(* PLC project TemplatePLC210_01, CODESYS CODESYS V3.5 SP17 Patch 3 *)
(* stored: creationDateTime 2025-07-22T12:00:36.9424136, version 3.5.14.30, modificationDateTime 2025-07-22T12:00:25.3757324, organization Production association OWEN *)

TYPE TRG_LeftSide :
STRUCT
	xFastDi01:				BOOL;
	xFastDi02:				BOOL;
	xFastDi03:				BOOL;
	xFastDi04:				BOOL;
	xFastDi05:				BOOL;
	xFastDi06:				BOOL;
	xFastDi07:				BOOL;
	xFastDi08:				BOOL;
	xFastDi09: 				BOOL;
	xFastDi10:				BOOL;
	xFastDi11:				BOOL;
	xFastDi12:				BOOL;
	
	xDo01:					BOOL;
	xDo02:					BOOL;
	xDo03:					BOOL;
	xDo04:					BOOL;
	
	udiCounterFastDi01:		UDINT;
	udiCounterFastDi02:		UDINT;
	udiCounterFastDi03:		UDINT;
	udiCounterFastDi04:		UDINT;
	udiCounterFastDi05:		UDINT;
	udiCounterFastDi06:		UDINT;
	udiCounterFastDi07:		UDINT;
	udiCounterFastDi08:		UDINT;
	udiCounterFastDi09:		UDINT;
	udiCounterFastDi10:		UDINT;
	udiCounterFastDi11:		UDINT;
	udiCounterFastDi12:		UDINT;
	
	udiPulseDurationFastDi01:	UDINT;
	udiPulseDurationFastDi02:	UDINT;
	udiPulseDurationFastDi03:	UDINT;
	udiPulseDurationFastDi04:	UDINT;
	udiPulseDurationFastDi05:	UDINT;
	udiPulseDurationFastDi06:	UDINT;
	udiPulseDurationFastDi07:	UDINT;
	udiPulseDurationFastDi08:	UDINT;
	udiPulseDurationFastDi09:	UDINT;
	udiPulseDurationFastDi10:	UDINT;
	udiPulseDurationFastDi11:	UDINT;
	udiPulseDurationFastDi12:	UDINT;

	udiPulsePeriodFastDi01:		UDINT;
	udiPulsePeriodFastDi02:		UDINT;
	udiPulsePeriodFastDi03:		UDINT;
	udiPulsePeriodFastDi04:		UDINT;
	udiPulsePeriodFastDi05:		UDINT;
	udiPulsePeriodFastDi06:		UDINT;
	udiPulsePeriodFastDi07:		UDINT;
	udiPulsePeriodFastDi08:		UDINT;
	udiPulsePeriodFastDi09:		UDINT;
	udiPulsePeriodFastDi10:		UDINT;
	udiPulsePeriodFastDi11:		UDINT;
	udiPulsePeriodFastDi12:		UDINT;
	
	udiGenPulseCountDo01:	    UDINT;
	udiGenPulseCountDo02:	    UDINT;
	udiGenPulseCountDo03:	    UDINT;
	udiGenPulseCountDo04:	    UDINT;
	
	udiGenPulseCountLeftDo01:	UDINT;
	udiGenPulseCountLeftDo02:	UDINT;
	udiGenPulseCountLeftDo03:	UDINT;
	udiGenPulseCountLeftDo04:	UDINT;
	
	udiPwmDutyCycleDo01:		UDINT;
	udiPwmDutyCycleDo02:		UDINT;
	udiPwmDutyCycleDo03:		UDINT;
	udiPwmDutyCycleDo04:		UDINT;
	
	diPulseCounterAbEncoder01: DINT;
	diPulseCounterAbEncoder02: DINT;
	diPulseCounterAbEncoder03: DINT;
	diPulseCounterAbEncoder04: DINT;
	diPulseCounterAbEncoder05: DINT;
	diPulseCounterAbEncoder06: DINT;
	
	diPulseCounterAbzEncoder01: DINT;
	diPulseCounterAbzEncoder02: DINT;
	diPulseCounterAbzEncoder03: DINT;
	
	diTurnCounterAbzEncoder01: DINT;
	diTurnCounterAbzEncoder02: DINT;
	diTurnCounterAbzEncoder03: DINT;
END_STRUCT
END_TYPE

TYPE TRG_Debug :
STRUCT
	xEnable: 			BOOL;
	udiPollingTime:		UDINT;
	udiRamUsedSize:		UDINT;
	udiRamFreeSize:		UDINT;
	udiCountHandles:	UDINT;
	udiProcUsage:		UDINT;
END_STRUCT
END_TYPE

TYPE TRG_Drives :
STRUCT
	xEnable:			BOOL;
	
	uliFsFullSize: 		ULINT;
	uliFsUsedSize: 		ULINT;
	uliFsFreeSize: 		ULINT;
	
	xUsbMounted:		BOOL;
	xUsbUnmount:		BOOL;
	xUsbUnmountDone:	BOOL;
	
	uliUsbFullSize: 	ULINT;
	uliUsbUsedSize: 	ULINT;
	uliUsbFreeSize: 	ULINT;
	
	xSdMounted:			BOOL;
	xSdUnmount:			BOOL;
	xSdUnmountDone:		BOOL;
	
	uliSdFullSize: 		ULINT;
	uliSdUsedSize: 		ULINT;
	uliSdFreeSize: 		ULINT;
END_STRUCT
END_TYPE

TYPE TRG_Info :
STRUCT
	sVendorName: 			STRING;
	sDeviceName: 			STRING;
	sSerialId: 				STRING;
	sRuntimeVersion:		STRING;
	sFirmwareVersion: 		STRING;
	sLinuxVersion: 			STRING;
	sNeedTargetVersion:		STRING;
	
	sProjectName:			STRING;
	sAuthorName:			STRING;
	sProjectVersion:		STRING;
	sProjectProfile:		STRING;
	dtProjectLastChanges:	DT;
END_STRUCT
END_TYPE

TYPE TRG_PLC210 :
STRUCT
	xPowerInput1:	  BOOL;
	xPowerInput2: 	  BOOL;
	xServiceButton:   BOOL;
	rCpuTemp:		  REAL;
	xStartStopSwitch: BOOL;
END_STRUCT
END_TYPE

TYPE TRG_RTC :
STRUCT
	uiGetYear:			UINT;
	usiGetMonth:		USINT;
	usiGetDay:			USINT;
	usiGetHour:			USINT;
	usiGetMinute:		USINT;
	usiGetSecond:		USINT;
	usiGetDayOfWeek:	USINT;
	usiGetWeekOfYear:	USINT;
	sGetFormatDate:		STRING;
	sGetFormatTime:		STRING;
	siGetUtcOffset:		SINT;
	dtDateAndTime:		DT;
	
	
	uiSetYear:			UINT;
	usiSetMonth:		USINT;
	usiSetDay:			USINT;
	usiSetHour:			USINT;
	usiSetMinute:		USINT;
	usiSetSecond:		USINT;
	siSetUtcOffset:		SINT;
	xUpdateSettings:	BOOL;
	
	xEnableNtp:			BOOL;
	xIsNtpEnabled:		BOOL;
	sPreferNtpServer:	STRING;
	usiNtpErrorCode:	USINT;
	
	ltSystemTick:		LTIME;
END_STRUCT
END_TYPE

TYPE TRG_Watchdog :
STRUCT
	eHandlingType:						Watchdog.ExceptionHandling;
	udiLastExceptionCode:				UDINT;
	sLastExceptionText:					STRING;
	dtLastExceptionTime:				DT;
	xIsHardwareWatchdogReboot:			BOOL;
	xDoReboot:							BOOL;
	usiPowerRebootCount:				USINT;
	usiExceptionRebootCount:			USINT;
	usiCommandRebootCount:				USINT;
	usiHardwareWatchdogRebootCount:		USINT;
	xResetCounters:						BOOL;
END_STRUCT
END_TYPE

TYPE TRG_RightSide :
STRUCT
	xSystemBusLink:				  BOOL;
	udiSystemBusError:  		  UDINT;
	
	xDo05:						  BOOL;
	xDo06:						  BOOL;
	xDo07:						  BOOL;
	xDo08:						  BOOL;
	xDo09:						  BOOL;
	xDo10:						  BOOL;
	xDo11:						  BOOL;
	xDo12:						  BOOL;

	xWriteAllAiSettings:  		  BOOL;
	
	xWriteSettingsAi1:	  		  BOOL;
	eWriteSensorTypeAi1:		  Mx210Assistant.ANALOG_SENSORS;
	rWriteOffsetAi1:			  REAL;
	rWriteMulAi1:			 	  REAL;
	rWriteHighLimitAi1:		 	  REAL;
	rWriteLowLimitAi1:		 	  REAL;
	uiWriteFilterBandAi1:	  	  UINT;
	uiWriteFilterTimeAi1:	  	  UINT;
	
	xWriteSettingsAi2:	  		  BOOL;
	eWriteSensorTypeAi2:		  Mx210Assistant.ANALOG_SENSORS;
	rWriteOffsetAi2:			  REAL;
	rWriteMulAi2:			 	  REAL;
	rWriteHighLimitAi2:		  	  REAL;
	rWriteLowLimitAi2:		  	  REAL;
	uiWriteFilterBandAi2:	  	  UINT;
	uiWriteFilterTimeAi2:	  	  UINT;
	
	xWriteSettingsAi3:	  		  BOOL;
	eWriteSensorTypeAi3:		  Mx210Assistant.ANALOG_SENSORS;
	rWriteOffsetAi3:			  REAL;
	rWriteMulAi3:			 	  REAL;
	rWriteHighLimitAi3:		  	  REAL;
	rWriteLowLimitAi3:		  	  REAL;
	uiWriteFilterBandAi3:	  	  UINT;
	uiWriteFilterTimeAi3:	  	  UINT;
	
	xWriteSettingsAi4:	  		  BOOL;
	eWriteSensorTypeAi4:		  Mx210Assistant.ANALOG_SENSORS;
	rWriteOffsetAi4:			  REAL;
	rWriteMulAi4:			 	  REAL;
	rWriteHighLimitAi4:		  	  REAL;
	rWriteLowLimitAi4:		  	  REAL;
	uiWriteFilterBandAi4:	  	  UINT;
	uiWriteFilterTimeAi4:	  	  UINT;
	
	xReadAllAiSettings:  		  BOOL;
	
	xReadSettingsAi1:	  		  BOOL;
	eReadSensorTypeAi1:		  	  Mx210Assistant.ANALOG_SENSORS;
	rReadOffsetAi1:			  	  REAL;
	rReadMulAi1:			 	  REAL;
	rReadHighLimitAi1:		 	  REAL;
	rReadLowLimitAi1:		 	  REAL;
	uiReadFilterBandAi1:	  	  UINT;
	uiReadFilterTimeAi1:	  	  UINT;
	
	xReadSettingsAi2:	  		  BOOL;
	eReadSensorTypeAi2:		  	  Mx210Assistant.ANALOG_SENSORS;
	rReadOffsetAi2:			  	  REAL;
	rReadMulAi2:			 	  REAL;
	rReadHighLimitAi2:		  	  REAL;
	rReadLowLimitAi2:		  	  REAL;
	uiReadFilterBandAi2:	  	  UINT;
	uiReadFilterTimeAi2:	  	  UINT;
	
	xReadSettingsAi3:	  		  BOOL;
	eReadSensorTypeAi3:		  	  Mx210Assistant.ANALOG_SENSORS;
	rReadOffsetAi3:			  	  REAL;
	rReadMulAi3:			 	  REAL;
	rReadHighLimitAi3:		  	  REAL;
	rReadLowLimitAi3:		  	  REAL;
	uiReadFilterBandAi3:	  	  UINT;
	uiReadFilterTimeAi3:	  	  UINT;
	
	xReadSettingsAi4:	  		  BOOL;
	eReadSensorTypeAi4:		  	  Mx210Assistant.ANALOG_SENSORS;
	rReadOffsetAi4:			  	  REAL;
	rReadMulAi4:			 	  REAL;
	rReadHighLimitAi4:		  	  REAL;
	rReadLowLimitAi4:		  	  REAL;
	uiReadFilterBandAi4:	  	  UINT;
	uiReadFilterTimeAi4:	  	  UINT;
	
	rValueAi1:					  REAL;
	uiTimeAi1:					  UINT;
	eStatusAi1:					  Mx210Assistant.ANALOG_SENSOR_ERRORS;
	
	rValueAi2:					  REAL;
	uiTimeAi2:					  UINT;
	eStatusAi2:					  Mx210Assistant.ANALOG_SENSOR_ERRORS;

	rValueAi3:					  REAL;
	uiTimeAi3:					  UINT;
	eStatusAi3:					  Mx210Assistant.ANALOG_SENSOR_ERRORS;

	rValueAi4:					  REAL;
	uiTimeAi4:					  UINT;
	eStatusAi4:					  Mx210Assistant.ANALOG_SENSOR_ERRORS;	
END_STRUCT
END_TYPE

TYPE TRG_Buzzer :
STRUCT
	xGet:	BOOL;
	xSet:	BOOL;
END_STRUCT
END_TYPE

TYPE VFD :
STRUCT
	irMaxFreq : REAL := 50;					
	irUpdateCycleStep : REAL := 1.5;
	irActualFreqInaccuracy : REAL := 0.2;
	
	iqISetFreq : UINT;
	
	itUpdateCycle : TIME := T#2S;
	
	ixStart : BOOL;
	ixChange : BOOL;
	ixStop : BOOL;
	ixReset : BOOL;
	ixSmoothStop : BOOL;
	ixEmergencyStop : BOOL;
	
	ixStarted : BOOL;
	ixStopped : BOOL;
	
	qxEmergencyStopStatus : BOOL;
	qxStartStatus : BOOL;
	qxStopStatus : BOOL;
	qxErrorInvalidInaccuracy : BOOL;
	qxDeviceError : BOOL;
	qxDelayError : BOOL;
END_STRUCT
END_TYPE

TYPE varAuto :
STRUCT
	Auto_ixFrqStart : BOOL;
	Auto_ixFrqChange : BOOL;
	Auto_ixFrqStop : BOOL;
	Auto_ixFrqEmergencyStop : BOOL;
	Auto_ixFrqReset : BOOL;
	Auto_ixFrqSmoothStop : BOOL;
	
	Auto_iqrSetFreq : REAL;
	
	Auto_ixKM_PU01 : BOOL;
	Auto_ixKM_PU02 : BOOL;
	Auto_ixKM_PU03 : BOOL;
	Auto_ixKM_PU04 : BOOL;
	Auto_ixKM_PU05 : BOOL;
END_STRUCT
END_TYPE

TYPE cmdAuto :
STRUCT
	vfdMain_ixStart : BOOL;
	vfdMain_ixFastStart : BOOL;
	vfdMain_ixStop : BOOL;
	vfdMain_ixEmergencyStop : BOOL;
	vfdMain_ixReset : BOOL;
	
	vfdReserve_ixStart : BOOL;
	vfdReserve_ixFastStart : BOOL;
	vfdReserve_ixStop : BOOL;
	vfdReserve_ixEmergencyStop : BOOL;
	vfdReserve_ixReset : BOOL;
END_STRUCT
END_TYPE

INTERFACE IShutterCommands
METHOD cmdOpen : BOOL
VAR_INPUT
	xOpen : BOOL;
END_VAR
END_METHOD
METHOD cmdClose : BOOL
VAR_INPUT
	xClose : BOOL;
END_VAR
END_METHOD
METHOD cmdStop : BOOL
VAR_INPUT
	xStop : BOOL;
END_VAR
END_METHOD
METHOD cmdReset : BOOL
VAR_INPUT
	xReset : BOOL;
END_VAR
END_METHOD
END_INTERFACE

INTERFACE IShutterFeedback
METHOD GetStatusReady : BOOL
VAR_INPUT
	xReady : BOOL;
END_VAR
END_METHOD
METHOD GetStatusClosed : BOOL
VAR_INPUT
	xClosed : BOOL;
END_VAR
END_METHOD
METHOD GetStatusOpen : BOOL
VAR_INPUT
	xOpened : BOOL;
END_VAR
END_METHOD
METHOD GetStatusManual : BOOL
VAR_INPUT
	xManual : BOOL;
END_VAR
END_METHOD
METHOD GetStatusCommonError : BOOL
VAR_INPUT
	xCommonError : BOOL;
END_VAR
END_METHOD
END_INTERFACE

TYPE REAL_TO_2WORD : UNION
  rVar : REAL;
  wVar : ARRAY[0..1] OF WORD;
END_UNION;
END_TYPE

FUNCTION_BLOCK FB_SHUTTER_LEGACY
VAR_INPUT
	time_error_long_time_without_status : TIME; // Таймер проверки долгого ожидания сигнала
	ixready : BOOL; // Затвор готовность
	ixerror : BOOL; //Затвор ошибка (вход)
	ixopen : BOOL; // Сигнал на открытие затвора
	ixclose : BOOL; // Сигнал на закрытие затвора
	ixreset : BOOL; // Действие пользователя при возниковении ошибки / аварии
	ixopened_status : BOOL; // Статус от устройства на открытие затвора
	ixclosed_status : BOOL; // Статус от устройства на закрытие затвора
END_VAR
VAR_OUTPUT
	qxopen : BOOL; // Открыть затвор
	qxclose : BOOL; // Закрыть затвор
	qxerror_from_device : BOOL; // Затвор ошибка
	qxerror_long_time_without_status : BOOL; // Ошибка долгого ожидания ixready
	error_long_time_without_status_open_closed : BOOL; // Ошибка долгого ожидания статуса открыт/закрыт
	qxopened : BOOL; // Затвор открыт
	qxclosed : BOOL; // Затвор закрыт
	qxclose_process : BOOL; // Закрытие затвора в процессе
	qxopen_process : BOOL; // Закрытие затвора в процессе
END_VAR
VAR
	error_fixation : BOOL; // Фиксация положения при возникновении ошибки
	rtrig_open : R_TRIG;
	rtrig_close : R_TRIG;
	rtrig_ixopened_status : R_TRIG;
	rtrig_ixclosed_status : R_TRIG;
	rtrig_ixreset : R_TRIG;
	rtrig_ixerror : R_TRIG;
	ftrig_ixopened_status : F_TRIG;
	ftrig_ixclosed_status : F_TRIG;
	
	// Таймеры на открытие/закрытие
	delay_qxopen : TON;
	delay_qxclose : TON;
	delay_time : TIME := T#2S;
	// Обработка ошибок долгого ожидания
	ton_error_long_time_without_status : TON;
	ton_error_long_time_without_status_open_closed : TON;
END_VAR

                    

// 	===	Обработка ошибок ===


// Сброс ошибок пользователем
rtrig_ixreset(CLK:= ixreset, Q=> );
IF rtrig_ixreset.Q THEN 
	error_fixation := FALSE; 
	qxerror_from_device := FALSE;
END_IF;

// Фиксация статуса ошибки
rtrig_ixerror(CLK:= ixerror, Q=> );
IF 	rtrig_ixerror.Q
	OR qxerror_long_time_without_status
	THEN
		error_fixation := TRUE;
//		qxerror_long_time_without_status := FALSE;
END_IF;
IF rtrig_ixerror.Q THEN qxerror_from_device := TRUE; END_IF;
	
// Обработка ошибки длительного ожидания статуса открыт/закрыт
ton_error_long_time_without_status_open_closed(
	IN:= qxclose_process OR qxopen_process, 
	PT:= time_error_long_time_without_status, 
	Q=> error_long_time_without_status_open_closed, 
	ET=> );


// 	===	Работа открытия/закрытия ===


rtrig_open(CLK:= ixopen, Q=> );
rtrig_close(CLK:= ixclose, Q=> );

rtrig_ixopened_status(CLK:= ixopened_status, Q=> );
rtrig_ixclosed_status(CLK:= ixclosed_status, Q=> );

ftrig_ixopened_status(CLK:= ixopened_status, Q=> );
ftrig_ixclosed_status(CLK:= ixclosed_status, Q=> );

delay_qxopen(IN:= qxopen, PT:= delay_time, Q=> , ET=> );
delay_qxclose(IN:= qxclose, PT:= delay_time, Q=> , ET=> );

IF rtrig_ixopened_status.Q THEN 
	qxopened := TRUE; 
	qxopen_process := FALSE;
	qxopen := FALSE;
END_IF;
IF rtrig_ixclosed_status.Q THEN 
	qxclosed := TRUE; 
	qxclose_process := FALSE;
	qxclose := FALSE;
END_IF;

IF ftrig_ixopened_status.Q THEN qxopened := FALSE; END_IF;
IF ftrig_ixclosed_status.Q THEN qxclosed := FALSE; END_IF;

IF 	rtrig_open.Q 
	AND ixready
	AND NOT qxclose 
	AND NOT error_fixation
	AND NOT qxopen_process
	THEN
		qxopen := TRUE;
		qxopen_process:= TRUE;
END_IF;

// IF delay_qxopen.Q THEN qxopen := FALSE; END_IF;


IF 	rtrig_close.Q 
	AND ixready
	AND NOT qxopen
	AND NOT error_fixation
	AND NOT qxclose_process
	THEN
		qxclose := TRUE;
		qxclose_process := TRUE;
END_IF;

// IF delay_qxclose.Q THEN qxclose := FALSE; END_IF;
                  
END_FUNCTION_BLOCK

FUNCTION_BLOCK INPUT_OUTPUT

VAR_INPUT
	ixSignal : BOOL; // Входной сигнал
	itInputTime : TIME; // Время дребезга сигнала (максимальное значение)
	itRattling_count_reset : TIME; // Время обнуления счётчика получения сигнала (дребезг)
	ixResetAlarm : BOOL; // Сброс ошибки (дребезг)
END_VAR

VAR_OUTPUT
	qxSignal : BOOL; // Выходной сигнал
	qxRattlingAlarm : BOOL; // Выход ошибки (дребезг)
END_VAR

VAR
	rtrig_ixSignal : R_TRIG;
	rtrig_qxRattlingAlarm : R_TRIG;
	ton_SignalDelay : TON;
	tof_FSignalDelay : TOF;
	ton_rattling_count_reset : TON;
	ctu_rattling : CTU;
END_VAR

                    ton_SignalDelay(
	IN:= ixSignal, 
	PT:= itInputTime, 
	Q=> qxSignal, 
	ET=> );

tof_FSignalDelay(
	IN:= ton_SignalDelay.Q, 
	PT:= itInputTime, 
	Q=> qxSignal, 
	ET=> );
	
rtrig_ixSignal(CLK:= ixSignal, Q=> );	
rtrig_qxRattlingAlarm(CLK:= ctu_rattling.Q, Q=> );

IF rtrig_qxRattlingAlarm.Q THEN qxRattlingAlarm := TRUE; END_IF;

ctu_rattling(
	CU:= rtrig_ixSignal.Q, 
	RESET:= ton_rattling_count_reset.Q, 
	PV:= RATTLING_FUN(itTime:= itRattling_count_reset), 
	Q=> , 
	CV=> );
	
ton_rattling_count_reset(
	IN:= NOT ton_rattling_count_reset.Q, 
	PT:= itRattling_count_reset, 
	Q=> , 
	ET=> );
                  
END_FUNCTION_BLOCK

FUNCTION_BLOCK DEBUG_RATTLING
VAR_INPUT
	ixWork : BOOL;
	ixSignalFrequency : INT;
END_VAR
VAR_OUTPUT
	qxSignal : BOOL;
END_VAR
VAR
	signal : BOOL;
	ton_Rattling : TON;
	tof_Rattling : TOF;
	tSignalTime : TIME;
END_VAR

                    tSignalTime := INT_TO_TIME(1000 / ixSignalFrequency);
qxSignal := signal AND ixWork;

ton_Rattling(
	IN:= NOT ton_Rattling.Q, 
	PT:= tSignalTime, 
	Q=> signal, 
	ET=> );
// tof_Rattling(
// 	IN:= ton_Rattling.Q,
// 	PT:= tSignalTime, 
// 	Q=> signal, 
// 	ET=> );

		
                  
END_FUNCTION_BLOCK

FUNCTION RATTLING_FUN : INT
VAR_INPUT
	itTime : TIME;
END_VAR
VAR
	iTime : INT;
END_VAR

                    iTime := TIME_TO_INT(itTime);

IF iTime >= 0 THEN
	RATTLING_FUN := iTime / 95;
END_IF;
                  
END_FUNCTION

FUNCTION_BLOCK FB_FRQ_CTRL
VAR_INPUT
	irMaxFreq : REAL; // Максимальное значение частоты
	ixStart : BOOL; // Запуск
	ixChange : BOOL; // Переключение с байпас на ЧРП (старт контактора без плавного пуска)
	ixStop : BOOL; // Остановка
	ixEmergencyStop : BOOL; // Аварийная остановка
	itUpdateCycle : TIME; // Время обновления цикла смены частоты
	itCmdDelayTime : TIME; // Время задержки выключения выходных сигналов
	irUpdateCycleStep : REAL; // Шаг изменения частоты за 1 цикл itUpdateCycle
	irActualFreq : REAL; // Показания текущей частоты устройства
	irActualFreqInaccuracy : REAL; // Погрешность показаний частоты устройства
	ixDeviceReady : BOOL; // Готовность исполнительного механизма
	ixDeviceReserve : BOOL; // True - статус механизма - РЕЗЕРВНЫй
	ixDeviceReserveOn: BOOL; // True - при условии статуса РЕЗЕРВ, переключение работы на текущий механизм
	ixDeviceError : BOOL; // Ошибка исполнительного механизма
	ixReset : BOOL; // Сброс ошибок и аварийной остановки
	ixSmoothStop : BOOL; // Режим плавной остановки\
	ixStarted : BOOL; // Получение сигнала о старте механизма
	ixStopped : BOOL; // Получение сигнала о стопе механизма
END_VAR
VAR_OUTPUT
	qrFreq : REAL; // Задание частоты на выход
	qxEmergencyStopStatus : BOOL; // Статус аварийной остановки
	qxStart : BOOL; // Запуск исполнительного механизма
	qxStartStatus : BOOL; // Статус запущен
	qxStop : BOOL; // Остановка исполнительного механизма
	qxStopStatus : BOOL; // Статус остановлен
	qxErrorInvalidInaccuracy : BOOL; // Ошибка большой погрешности
	qxDeviceError : BOOL; // Ошибка исполнительного механизма (выход через блок)
	qxDelayError : BOOL; // Ошибка долгого ожидания обратной связи механизма после выполнения команды
END_VAR
VAR_IN_OUT
	iqrSetFreq : REAL; // Задание частоты на вход
END_VAR
VAR
	rtrig_ixStart : R_TRIG;
	rtrig_ixChange : R_TRIG;
	rtrig_ixStop : R_TRIG;
	rtrig_ixEmergencyStop : R_TRIG;
	rtrig_updateCycle : R_TRIG;
	rtrig_qxDeviceError : R_TRIG;
	rtrig_ixReset : R_TRIG;
	ftrig_stopPulse : F_TRIG;
	blink_updateCycle : BLINK;
	xWorkProcess : BOOL;
	xPossibleInac : BOOL;
	xErrorFixation : BOOL;
	ton_stopWorkProcess : TON;
	ton_qxStopDisable : TON;
	ton_qxStartDisable : TON;	
	reserve_iqrSetFreq : REAL;
END_VAR

                    rtrig_ixStart(CLK:= ixStart, Q=> );
rtrig_ixChange(CLK:= ixChange, Q=> );
rtrig_ixStop(CLK:= ixStop, Q=> );
rtrig_ixEmergencyStop(CLK:= ixEmergencyStop, Q=> );
rtrig_updateCycle(CLK:= blink_updateCycle.OUT, Q=> );
ftrig_stopPulse(CLK:= qrFreq > 0, Q=> );
rtrig_qxDeviceError(CLK:= ixDeviceError, Q=> );
rtrig_ixReset(CLK:= ixReset, Q=> );

IF ftrig_stopPulse.Q OR rtrig_ixEmergencyStop.Q THEN
	qxStop := TRUE;
ELSIF ixStopped THEN
	qxStop := FALSE;
ELSIF ton_qxStopDisable.Q THEN
	qxStop := FALSE;
	qxDelayError := TRUE;
END_IF;

IF (rtrig_ixStart.Q OR rtrig_ixChange.Q) AND NOT qxEmergencyStopStatus AND NOT xErrorFixation AND ixDeviceReady THEN
	qxStart := TRUE;
ELSIF ixStarted THEN
	qxStart := FALSE;
ELSIF ton_qxStartDisable.Q THEN
	qxStart := FALSE;
	qxDelayError := TRUE;
END_IF;

ton_qxStopDisable(
	IN:= qxStop, 
	PT:= itCmdDelayTime, 
	Q=> , 
	ET=> );

ton_qxStartDisable(
	IN:= qxStart, 
	PT:= itCmdDelayTime, 
	Q=> , 
	ET=> );

blink_updateCycle(
	ENABLE:= xWorkProcess, 
	TIMELOW:= itUpdateCycle, 
	TIMEHIGH:= T#100MS,
	OUT=> );

ton_stopWorkProcess(
	IN:= xWorkProcess AND qrFreq = 0, 
	PT:= T#5S, 
	Q=> , 
	ET=> );

IF NOT FC_PossibleInac(actualFreq:= irActualFreq, actualFreqInaccuracy:= irActualFreqInaccuracy, orderFreq:= qrFreq) THEN
	qxErrorInvalidInaccuracy := TRUE;
END_IF;
 
IF rtrig_qxDeviceError.Q THEN
	qxDeviceError := TRUE;
END_IF;
 
IF	qxErrorInvalidInaccuracy 
	OR qxDeviceError THEN
		xErrorFixation := TRUE;
END_IF;

IF rtrig_ixReset.Q THEN
	xErrorFixation := FALSE;
	qxEmergencyStopStatus := FALSE;
	qxErrorInvalidInaccuracy := FALSE;
	qxDeviceError := FALSE;
END_IF;
 
IF ton_stopWorkProcess.Q AND (NOT qxStopStatus OR NOT qxStartStatus) THEN 
	xWorkProcess := 0; 
	qxStopStatus := FALSE; 
	qxStartStatus := FALSE; 
END_IF;
IF rtrig_ixStart.Q AND ixDeviceReady AND (NOT xErrorFixation AND NOT qxEmergencyStopStatus) THEN 
	xWorkProcess := TRUE; 
	qxStartStatus := TRUE; 
	qxStopStatus := FALSE; 
END_IF;
IF rtrig_ixChange.Q AND ixDeviceReady AND (NOT xErrorFixation AND NOT qxEmergencyStopStatus) THEN
	xWorkProcess := TRUE; 
	qxStartStatus := TRUE; 
	qxStopStatus := FALSE;
	qrFreq := iqrSetFreq;
END_IF;
IF rtrig_ixStop.Q AND (NOT xErrorFixation AND NOT qxEmergencyStopStatus) THEN 
	reserve_iqrSetFreq := iqrSetFreq;
	iqrSetFreq := 0; 
	qxStopStatus := TRUE;  
	qxStartStatus := FALSE; 
	IF NOT ixSmoothStop THEN qrFreq := 0; END_IF;
END_IF;
IF ftrig_stopPulse.Q THEN iqrSetFreq := reserve_iqrSetFreq; xWorkProcess := 0; END_IF;
IF rtrig_ixEmergencyStop.Q THEN 
	xWorkProcess :=0;
	qrFreq := 0;
	qxEmergencyStopStatus := TRUE; 
	qxStopStatus := FALSE; 
	qxStartStatus := FALSE;
END_IF;

IF 	iqrSetFreq <> qrFreq 
	AND rtrig_updateCycle.Q 
	AND FC_PossibleInac(actualFreq:= irActualFreq, actualFreqInaccuracy:= irActualFreqInaccuracy, orderFreq:= qrFreq)
	AND ixDeviceReady
	AND NOT qxEmergencyStopStatus
	AND NOT xErrorFixation
	AND (iqrSetFreq <= irMaxFreq AND iqrSetFreq >= 0) THEN
		IF iqrSetFreq + irUpdateCycleStep < qrFreq THEN
			qrFreq := qrFreq - irUpdateCycleStep;
		ELSIF iqrSetFreq - irUpdateCycleStep > qrFreq THEN
			qrFreq := qrFreq + irUpdateCycleStep;
		ELSE
			qrFreq := iqrSetFreq;
		END_IF;
END_IF;
                  
END_FUNCTION_BLOCK

FUNCTION FC_PossibleInac : BOOL
VAR_INPUT
	actualFreq : REAL;
	actualFreqInaccuracy : REAL;
	orderFreq : REAL;
END_VAR
VAR
END_VAR

                    IF actualFreq < orderFreq THEN
	FC_PossibleInac := orderFreq - actualFreq <= actualFreqInaccuracy;
ELSIF actualFreq > orderFreq THEN
	FC_PossibleInac :=actualFreq - orderFreq <= actualFreqInaccuracy;
ELSIF actualFreq = orderFreq THEN
	FC_PossibleInac := TRUE;
ELSE
	RETURN;
END_IF;
                  
END_FUNCTION

FUNCTION_BLOCK FB_DEBUG_SET_ACTUAL_FREQ
VAR_INPUT
	irOrderFreq : REAL; // Задание частоты от блока FB_FRQ_CRTL
	irInac : REAL; // Значение погрешности
	itDelay : TIME; // Задержка сигнала на выход
	ixReverseInac : BOOL; // Если true, выходной сигнал равен  irOrderFreq - irInac, иначе irOrderFreq + irInac
END_VAR
VAR_OUTPUT
	qrActualFreq : REAL; // Выходной сигнал
END_VAR
VAR
	blink_signal : BLINK;
	rtrig_signal : R_TRIG;
END_VAR

                    blink_signal(
	ENABLE:= TRUE, 
	TIMELOW:= itDelay, 
	TIMEHIGH:= T#100MS, 
	OUT=> );

rtrig_signal(CLK:= blink_signal.OUT, Q=> );

IF rtrig_signal.Q AND ixReverseInac THEN
	qrActualFreq := irOrderFreq - irInac;
	
ELSE
	qrActualFreq := irOrderFreq + irInac;
END_IF;
                  
END_FUNCTION_BLOCK

FUNCTION_BLOCK FB_A_SIGNAL_SCALE
VAR_INPUT
	irSignal : REAL; 			// Вход аналогового сигнала
	irSignalSim : REAL; 		// Вход аналогового сигнала (симулятор)
	irSignalDownLimit : REAL; 	// Нижний предел сигнала
	irSignalUpLimit : REAL; 	// Верхний предел сигнала
	irValueDownLimit : REAL; 	// Нижний предел масштабированной единицы
	irValueUpLimit : REAL; 		// Верхий предел масштабированной единицы
	irHSignal : REAL; 			// Верхний предупредительный сигнал
	irHHSignal : REAL; 			// Верхний аварийный сигнал
	irLSignal : REAL; 			// Нижний предупредительный сигнал
	irLLSignall : REAL; 		// Верхний предупредительный сигнал
	ixReset : BOOL; 			// Ресет ошибок
	ixDeviceOn : BOOL; 			// Датчик работает
	ixSimulation : BOOL;		// Режим симуляции сигнала
END_VAR
VAR_OUTPUT
	qrSignal : REAL; 			// Выходной масштабированный сигнал
	qxMaxSignal : BOOL;			// Достижение минимального сигнала
	qxMinSignal : BOOL; 		// Достижение максимального сигнала
	qxErrorMin : BOOL; 			// Ошибка: сигнал меньше, чем минимально допустимый
	qxErrorMax : BOOL; 			// Ошибка: сигнал больше, чем максимально допустимый
	qxHSignal : BOOL; 			// Достижение верхнего предупредительного сигнала
	qxHHSignal : BOOL; 			// Достижение верхнего аварийного сигнала 
	qxLSignal : BOOL;			// Достижение нижнего предупредительного сигнала
	qxLLSignal : BOOL;			// Достижение нихнего аварийного сигнала
END_VAR
VAR
	rtrig_qxMaxSignal : R_TRIG;
	rtrig_qxMinSignal : R_TRIG;
	
	rtrig_qxErrorMin : R_TRIG;
	rtrig_qxErrorMax : R_TRIG;
	rtrig_ixReset : R_TRIG;
	
	rtrig_qxHSignal : R_TRIG;
	rtrig_qxHHSignal : R_TRIG;
	rtrig_qxLSignal : R_TRIG;
	rtrig_qxLLSignal : R_TRIG;
	
END_VAR

                    rtrig_ixReset(CLK:= ixReset, Q=> );

IF ixDeviceOn THEN
	rtrig_qxMaxSignal(CLK:= irSignal = irSignalUpLimit, Q=> );
	rtrig_qxMinSignal(CLK:= irSignal = irSignalDownLimit, Q=> );
	
	rtrig_qxErrorMax(CLK:= irSignal > irSignalUpLimit, Q=> );
	rtrig_qxErrorMin(CLK:= irSignal < irSignalDownLimit, Q=> );
	
	rtrig_qxHSignal(CLK:= irHSignal < qrSignal AND NOT qxHSignal, Q=> );
	rtrig_qxHHSignal(CLK:= irHHSignal < qrSignal AND NOT qxHHSignal, Q=> );
	rtrig_qxLSignal(CLK:= irLSignal > qrSignal AND NOT qxLSignal, Q=> );
	rtrig_qxLLSignal(CLK:= irLLSignall > qrSignal AND NOT qxLLSignal, Q=> );

	IF NOT qxErrorMin AND NOT qxErrorMax AND NOT ixSimulation THEN 
		qrSignal := ((irSignal - irSignalDownLimit) * (irValueUpLimit - irValueDownLimit)) / (irSignalUpLimit - irSignalDownLimit) + irValueDownLimit;
	END_IF;
	
ELSIF NOT qxErrorMin AND NOT qxErrorMax AND ixSimulation THEN
	qrSignal := ((irSignalSim - irSignalDownLimit) * (irValueUpLimit - irValueDownLimit)) / (irSignalUpLimit - irSignalDownLimit) + irValueDownLimit;
ELSE
	qrSignal := 0;
END_IF;

IF rtrig_qxHSignal.Q THEN qxHSignal := TRUE; END_IF;
IF rtrig_qxHHSignal.Q THEN qxHHSignal := TRUE; END_IF;
IF rtrig_qxLSignal.Q THEN qxLSignal := TRUE; END_IF;
IF rtrig_qxLLSignal.Q THEN qxLLSignal := TRUE; END_IF;

IF rtrig_ixReset.Q THEN
	qxHSignal := FALSE;
	qxHHSignal := FALSE;
	qxLSignal := FALSE;
	qxLLSignal := FALSE;
END_IF;

IF rtrig_qxMaxSignal.Q THEN qxMaxSignal := TRUE; END_IF;
IF rtrig_qxMinSignal.Q THEN qxMinSignal := TRUE; END_IF;
IF rtrig_qxErrorMax.Q THEN qxErrorMax := TRUE; END_IF;
IF rtrig_qxErrorMin.Q THEN qxErrorMin := TRUE; END_IF;

IF rtrig_ixReset.Q THEN
		qxMaxSignal := FALSE;
		qxMinSignal := FALSE;
		qxErrorMax := FALSE;
		qxErrorMin := FALSE;
END_IF;
                  
END_FUNCTION_BLOCK

FUNCTION_BLOCK FB_Contactor
VAR_INPUT
	ixStart : BOOL;
	ixStop : BOOL;
END_VAR
VAR_OUTPUT
	qxSignal : BOOL;
	qxStartStatus : BOOL;
	qxStopStatus : BOOL;
END_VAR
VAR
	rs_qxSignal : RS;
END_VAR

                    rs_qxSignal(SET:= ixStart, RESET1:= ixStop, Q1=> qxSignal);

qxStartStatus := qxSignal;
qxStopStatus := NOT qxSignal;
                  
END_FUNCTION_BLOCK

FUNCTION_BLOCK FB_SmStart
VAR_INPUT
	ixStart : BOOL;					// Пуск УПП
	ixStop : BOOL;					// Остановка УПП
	ixError : BOOL;					// Получение ошибки от устройства
	ixWorkProcess : BOOL;			// Получение статуса работы от устройства
	itStartTime : TIME;				// Время старта, заданное на устройстве
	itStopTime : TIME;				// Время остановки, заданное на устройстве
END_VAR
VAR_OUTPUT
	qxSignal : BOOL;				// Выходной сигнал на УПП
	qxError : BOOL;					// Выход из блока со статусом ошибки от устройства
	qxWorkProcess : BOOL;			// Выход из блока со статусом работы от устройства
	qxStartStatus : BOOL;			// Статус: УПП закончил работу и запущен
	qxStartProcess : BOOL;			// Статус: УПП в процессе старта
	qxStopStatus : BOOL;			// Статус: УПП закончил работу и остановлен
	qxStopProcess : BOOL;			// Статус: УПП в процессе остановки
END_VAR
VAR
	rtrig_ixStart : R_TRIG;
	ftrig_qxStartStatus : F_TRIG;
	tof_StartProcess : TOF;
	xStartProcess : BOOL;
	
	rtrig_ixStop : R_TRIG;
	ftrig_qxStopStatus : F_TRIG;
	tof_StopProcess : TOF;
	
	xStartCondition : BOOL;
	xStopCondition : BOOL;
END_VAR

                    qxWorkProcess := ixWorkProcess;
qxError := ixError;
xStartCondition := rtrig_ixStart.Q AND NOT ixError AND NOT qxStartStatus;
xStopCondition := rtrig_ixStop.Q AND NOT ixError AND NOT qxStopStatus;

// Работа на старт

rtrig_ixStart(CLK:= ixStart, Q=> );
ftrig_qxStartStatus(CLK:= tof_StartProcess.Q, Q=> );

tof_StartProcess(
	IN:= rtrig_ixStart.Q AND NOT ixError,
	PT:= itStartTime, 
	Q=> qxStartProcess, 
	ET=> );

IF xStartCondition THEN qxSignal := TRUE; qxStopProcess := FALSE; qxStopStatus := FALSE; END_IF;
IF ftrig_qxStartStatus.Q THEN qxStartStatus := TRUE; END_IF;

// Работа на стоп

rtrig_ixStop(CLK:= ixStop, Q=> );
ftrig_qxStopStatus(CLK:= tof_StopProcess.Q, Q=> );

tof_StopProcess(
	IN:= rtrig_ixStop.Q AND NOT ixError, 
	PT:= itStopTime, 
	Q=> qxStopProcess, 
	ET=> );
	
IF xStopCondition THEN qxSignal := FALSE; qxStartProcess := FALSE; qxStartStatus := FALSE; END_IF;
IF ftrig_qxStopStatus.Q THEN qxStopStatus := TRUE; END_IF;

                  
END_FUNCTION_BLOCK

FUNCTION_BLOCK FB_TEST_FRQ_CTRL
VAR_INPUT
	irMaxFreq : REAL; // Максимальное значение частоты
	ixStart : BOOL; // Запуск
	ixChange : BOOL; // Переключение с байпас на ЧРП (старт контактора без плавного пуска)
	ixStop : BOOL; // Остановка
	ixEmergencyStop : BOOL; // Аварийная остановка
	itUpdateCycle : TIME; // Время обновления цикла смены частоты
	itCmdDelayTime : TIME; // Время задержки выключения выходных сигналов
	irUpdateCycleStep : REAL; // Шаг изменения частоты за 1 цикл itUpdateCycle
	irActualFreq : REAL; // Показания текущей частоты устройства
	irActualFreqInaccuracy : REAL; // Погрешность показаний частоты устройства
	ixDeviceReady : BOOL; // Готовность исполнительного механизма
	ixDeviceReserve : BOOL; // True - статус механизма - РЕЗЕРВНЫй
	ixDeviceReserveOn: BOOL; // True - при условии статуса РЕЗЕРВ, переключение работы на текущий механизм
	ixDeviceError : BOOL; // Ошибка исполнительного механизма
	ixReset : BOOL; // Сброс ошибок и аварийной остановки
	ixSmoothStop : BOOL; // Режим плавной остановки\
	ixStarted : BOOL; // Получение сигнала о старте механизма
	ixStopped : BOOL; // Получение сигнала о стопе механизма
END_VAR
VAR_OUTPUT
	qrFreq : REAL; // Задание частоты на выход
	qxEmergencyStopStatus : BOOL; // Статус аварийной остановки
	qxStart : BOOL; // Запуск исполнительного механизма
	qxStartStatus : BOOL; // Статус запущен
	qxStop : BOOL; // Остановка исполнительного механизма
	qxStopStatus : BOOL; // Статус остановлен
	qxErrorInvalidInaccuracy : BOOL; // Ошибка большой погрешности
	qxDeviceError : BOOL; // Ошибка исполнительного механизма (выход через блок)
	qxDelayError : BOOL; // Ошибка долгого ожидания обратной связи механизма после выполнения команды
END_VAR
VAR_IN_OUT
	iqrSetFreq : REAL; // Задание частоты на вход
END_VAR
VAR
    // Триггеры и таймеры
    rtrig_ixStart : R_TRIG;
    rtrig_ixChange : R_TRIG;
    rtrig_ixStop : R_TRIG;
    rtrig_ixEmergencyStop : R_TRIG;
    rtrig_updateCycle : R_TRIG;
    rtrig_qxDeviceError : R_TRIG;
    rtrig_ixReset : R_TRIG;
    ftrig_stopPulse : F_TRIG;
    blink_updateCycle : BLINK;
    ton_stopWorkProcess : TON;
    ton_qxStopDisable : TON;
    ton_qxStartDisable : TON;
    
    // Внутренние состояния
    xWorkProcess : BOOL;
    xErrorFixation : BOOL;
    reserve_iqrSetFreq : REAL;
END_VAR

                    // Инициализация триггеров
rtrig_ixStart(CLK:= ixStart);
rtrig_ixChange(CLK:= ixChange);
rtrig_ixStop(CLK:= ixStop);
rtrig_ixEmergencyStop(CLK:= ixEmergencyStop);
ftrig_stopPulse(CLK:= qrFreq > 0);
rtrig_qxDeviceError(CLK:= ixDeviceError);
rtrig_ixReset(CLK:= ixReset);
rtrig_updateCycle(CLK:= blink_updateCycle.OUT);

// Основная логика
ProcessReset();
ProcessStartStopCommands();
ProcessFrequencyControl();
ProcessErrorHandling();
ProcessTimers();
                  

METHOD UpdateWorkStatus : BOOL
VAR_INPUT
END_VAR
                          // Сброс статусов при завершении
IF ton_stopWorkProcess.Q AND (NOT qxStopStatus OR NOT qxStartStatus) THEN 
    xWorkProcess := FALSE; 
    qxStopStatus := FALSE; 
    qxStartStatus := FALSE;
    RETURN;
END_IF;

// Обработка команд
CASE TRUE OF
    rtrig_ixStart.Q: 
        IF CheckStartConditions() THEN 
            xWorkProcess := TRUE; 
            qxStartStatus := TRUE;
        END_IF;
        
    rtrig_ixChange.Q: 
        IF CheckStartConditions() THEN 
            xWorkProcess := TRUE; 
            qxStartStatus := TRUE;
        END_IF;
        
    rtrig_ixStop.Q: 
        IF NOT xErrorFixation AND NOT qxEmergencyStopStatus THEN 
            reserve_iqrSetFreq := iqrSetFreq;
            iqrSetFreq := 0; 
            qxStopStatus := TRUE;
        END_IF;
        
    rtrig_ixEmergencyStop.Q: 
        xWorkProcess := FALSE;
        qxEmergencyStopStatus := TRUE;
END_CASE;
                        
END_METHOD

METHOD ShouldUpdateFrequency  : BOOL
VAR_INPUT
END_VAR
                          ShouldUpdateFrequency := iqrSetFreq <> qrFreq 
	AND rtrig_updateCycle.Q 
	AND CheckFrequencyInaccuracy()
	AND ixDeviceReady
	AND NOT qxEmergencyStopStatus
	AND NOT xErrorFixation
	AND (iqrSetFreq <= irMaxFreq) 
	AND (iqrSetFreq >= 0);
                        
END_METHOD

METHOD ProcessStopActions  : BOOL
VAR_INPUT
END_VAR
                          IF rtrig_ixStop.Q AND NOT xErrorFixation AND NOT qxEmergencyStopStatus THEN
    IF NOT ixSmoothStop THEN 
        qrFreq := 0; 
    END_IF;
ELSIF rtrig_ixEmergencyStop.Q THEN 
    qrFreq := 0;
ELSIF ftrig_stopPulse.Q THEN 
    iqrSetFreq := reserve_iqrSetFreq; 
    xWorkProcess := FALSE; 
END_IF;
                        
END_METHOD

METHOD ProcessFrequencyControl  : BOOL
VAR_INPUT
END_VAR
                          // Прямая установка частоты для CHANGE
IF rtrig_ixChange.Q AND CheckStartConditions() THEN
    qrFreq := iqrSetFreq;
END_IF;

// Плавное изменение частоты
IF ShouldUpdateFrequency() THEN
    qrFreq := CalculateNewFrequency();
END_IF;

// Обработка остановки и аварийных ситуаций
ProcessStopActions();
                        
END_METHOD

METHOD ProcessStartStopCommands : BOOL
VAR_INPUT
END_VAR
                          // Обработка команды STOP
IF ftrig_stopPulse.Q OR rtrig_ixEmergencyStop.Q THEN
	qxStop := TRUE;
ELSIF ixStopped THEN
	qxStop := FALSE;
ELSIF ton_qxStopDisable.Q THEN
	qxStop := FALSE;
	qxDelayError := TRUE;
END_IF;

// Обработка команды START
IF (rtrig_ixStart.Q OR rtrig_ixChange.Q) AND NOT qxEmergencyStopStatus AND NOT xErrorFixation AND ixDeviceReady THEN
	qxStart := TRUE;
ELSIF ixStarted THEN
	qxStart := FALSE;
ELSIF ton_qxStartDisable.Q THEN
	qxStart := FALSE;
	qxDelayError := TRUE;
END_IF;

// Обновление статусов работы
UpdateWorkStatus();
                        
END_METHOD

METHOD ProcessReset : BOOL
VAR_INPUT
END_VAR
                          IF rtrig_ixReset.Q THEN
    xErrorFixation := FALSE;
    qxEmergencyStopStatus := FALSE;
    qxErrorInvalidInaccuracy := FALSE;
    qxDeviceError := FALSE;
	qxDelayError := FALSE;
END_IF;
                        
END_METHOD

METHOD CheckStartConditions : BOOL
VAR_INPUT
END_VAR
                          CheckStartConditions := NOT qxEmergencyStopStatus  AND NOT xErrorFixation  AND ixDeviceReady;
                        
END_METHOD

METHOD CalculateNewFrequency  : REAL
VAR_INPUT
END_VAR
                          IF iqrSetFreq + irUpdateCycleStep < qrFreq THEN
	CalculateNewFrequency := qrFreq - irUpdateCycleStep;
ELSIF iqrSetFreq - irUpdateCycleStep > qrFreq THEN
	CalculateNewFrequency := qrFreq + irUpdateCycleStep;
ELSE
	CalculateNewFrequency := iqrSetFreq;
END_IF;
                        
END_METHOD

METHOD CheckFrequencyInaccuracy : BOOL
VAR_INPUT
END_VAR
                          IF irActualFreq < qrFreq THEN
	CheckFrequencyInaccuracy := qrFreq - irActualFreq <= irActualFreqInaccuracy;
ELSIF irActualFreq > qrFreq THEN
	CheckFrequencyInaccuracy :=irActualFreq - qrFreq <= irActualFreqInaccuracy;
ELSIF irActualFreq = qrFreq THEN
	CheckFrequencyInaccuracy := TRUE;
ELSE
	CheckFrequencyInaccuracy := FALSE;
END_IF;
                        
END_METHOD

METHOD ProcessErrorHandling : BOOL
VAR_INPUT
END_VAR
                          // Проверка погрешности частоты
qxErrorInvalidInaccuracy := NOT CheckFrequencyInaccuracy();

// Фиксация ошибок устройства
IF rtrig_qxDeviceError.Q THEN
    qxDeviceError := TRUE;
END_IF;

// Общая фиксация ошибок
xErrorFixation := qxErrorInvalidInaccuracy OR qxDeviceError;
                        
END_METHOD

METHOD ProcessTimers : BOOL
VAR_INPUT
END_VAR
                          // Таймеры для команд
ton_qxStopDisable(IN:= qxStop, PT:= itCmdDelayTime);
ton_qxStartDisable(IN:= qxStart, PT:= itCmdDelayTime);

// Таймер для цикла обновления
blink_updateCycle(
    ENABLE:= xWorkProcess, 
    TIMELOW:= itUpdateCycle, 
    TIMEHIGH:= T#100MS
);

// Таймер остановки рабочего процесса
ton_stopWorkProcess(
    IN:= xWorkProcess AND qrFreq = 0, 
    PT:= T#5S
);
                        
END_METHOD
END_FUNCTION_BLOCK

PROGRAM LEGACY_MAIN
VAR
	// 	== ДЛЯ ТЕСТА, ПОТОМ УДАЛИТЬ ==

	PLC_Mode : INT := 0; // 0 – «Авто», 1 – «Обрыв связи», 2 – «Местный-Сервис»
	
	// LeftSide Маска входов ПЛК
	_0303_05_PU01_ixKM_StatusOn : BOOL;				// Контактор ПРЯМ. ПУСК Насос 0303.05-PU-01
	_0303_05_PU01_ixKM_VFD_StatusOn : BOOL;			// Контактор ПРЯМ. ЧРП Насос 0303.05-PU-01
	_0303_05_PU02_ixKM_StatusOn : BOOL;				// Контактор ПРЯМ. ПУСК Насос 0303.05-PU-02
	_0303_05_PU02_ixKM_VFD_StatusOn : BOOL;			// Контактор ПРЯМ. ЧРП Насос 0303.05-PU-02
	_0303_05_PU03_ixKM_StatusOn : BOOL;				// Контактор ПРЯМ. ПУСК Насос 0303.05-PU-03
	_0303_05_PU03_ixKM_VFD_StatusOn : BOOL;			// Контактор ПРЯМ. ЧРП Насос 0303.05-PU-03
	_0303_05_PU04_ixKM_StatusOn : BOOL;				// Контактор ПРЯМ. ПУСК Насос 0303.05-PU-04
	_0303_05_PU04_ixKM_VFD_StatusOn : BOOL;			// Контактор ПРЯМ. ЧРП Насос 0303.05-PU-04
	_0303_05_PU05_ixKM_StatusOn : BOOL;				// Контактор ПРЯМ. ПУСК Насос 0303.05-PU-05
	_0303_05_PU05_ixKM_VFD_StatusOn : BOOL;			// Контактор ПРЯМ. ЧРП Насос 0303.05-PU-05
	_0303_05_BY08_ixShutter_PosOpen : BOOL;			// Положение ОТКР. Затвор 0303.05-BY-08
	_0303_05_BY08_ixShutter_PosClosed : BOOL;		// Положение ЗАКР. Затвор 0303.05-BY-08
	
	// RightSide Маска выходов ПЛК
	_0303_05_qxEmergencyStop : BOOL;			// Реле аварийного останова
	_0303_05_PU01_qxDryRun : BOOL;				// Насос 0303.05-PU-01 Сухой ход
	_0303_05_PU02_qxDryRun : BOOL;				// Насос 0303.05-PU-02 Сухой ход
	_0303_05_PU03_qxDryRun : BOOL;				// Насос 0303.05-PU-03 Сухой ход
	_0303_05_PU04_qxDryRun : BOOL;				// Насос 0303.05-PU-04 Сухой ход
	_0303_05_PU05_qxDryRun : BOOL;				// Насос 0303.05-PU-05 Сухой ход
	_0303_05_1KM8_qxOn : BOOL;					// Включить 1KM8
	_0303_05_2KM8_qxOn : BOOL;					// Включить 2KM8
	
	// 	==============================================
	
	// Общие глобальные переменные
	iIPU_Select : USINT; 			// Выбор насоса для старта
	ixKM_PU01 : BOOL; 				// Насос 1 переключение на байпас
	ixKM_PU02 : BOOL;				// Насос 2 переключение на байпас
	ixKM_PU03 : BOOL;				// Насос 3 переключение на байпас
	ixKM_PU04 : BOOL;				// Насос 4 переключение на байпас
	ixKM_PU05 : BOOL;				// Насос 5 переключение на байпас
	xKMFrqReady : BOOL;			
	xPuKmFrqWorked : BOOL;			// True - какой либо из насосов от ЧРП в работе
	xSimulationStatus : BOOL;		// True - включен режим симуляции с предварительными настройками (по стандарту режим ПЛК Auto)
	autoCmd : varAuto;					// Переменные для симуляции
	inputOutput_ButtonInputTime : TIME := T#100MS;
	ix1KM8_qxOn : BOOL;				// Включение контактора 1KM8
	ix2KM8_qxOn : BOOL;				// Включение контактора 2KM8
	ix1KM8_qxOff : BOOL;			// Выключение контактора 1KM8
	ix2KM8_qxOff: BOOL;				// Выключение контактора 2KM8
	// Обработка команд АСУТП и сервис
	_0303_05_CommandProceed : FB_CommandProceed;
	
	//inputOutput_Rattling : TIME := T#3S;
	
	//	VFD001 переменные и ФБ ЧРП
	VFD001 : FB_FRQ_CTRL;
	VFD002 : FB_FRQ_CTRL;
	RS_0303_05_PU01_qxKM_Frq_cmdOn : RS;
	RS_0303_05_PU02_qxKM_Frq_cmdOn : RS;
	RS_0303_05_PU03_qxKM_Frq_cmdOn : RS;
	RS_0303_05_PU04_qxKM_Frq_cmdOn : RS;
	RS_0303_05_PU05_qxKM_Frq_cmdOn : RS;
	
	varVFD001 : VFD;
	varVFD002 : VFD;
	
	VFD001_iqrSetFreq : REAL; // Переменная задания частоты
	
	VFD001_rtrig_ixStop : R_TRIG;
	VFD001_ixStopped : F_TRIG;
	VFD001_rtrig_ixStart : R_TRIG;
	VFD001_rtrig_ixChange : R_TRIG;
	VFD001_DebugActualFreqSim : FB_DEBUG_SET_ACTUAL_FREQ;
	VFD002_DebugActualFreqSim : FB_DEBUG_SET_ACTUAL_FREQ;
	VFD001_ton_StopDelay : TON;
	// Масштабирование сигнала ддя модуля аналогово выхода 
	SetFreqAnaloOutputSignalScale : FB_Asignal_FreqConvertation;
	
	
	// _0303_05_BY01 Затвор переменные ФБ
	_0303_05_BY01 : FB_SHUTTER_LEGACY;
	_0303_05_BY01_Contactor_PosOpen_FB : INPUT_OUTPUT;
	_0303_05_BY01_Contactor_PosClosed_FB : INPUT_OUTPUT;
	_0303_05_BY01_ixShutter_StatusReady_FB : INPUT_OUTPUT;
	_0303_05_BY01_ixShutter_StatusError_FB : INPUT_OUTPUT;
	_0303_05_BY01_ixShutter_PosOpen_FB : INPUT_OUTPUT;
	_0303_05_BY01_ixShutter_PosClosed_FB : INPUT_OUTPUT;
	_0303_05_BY01_ixreset : BOOL;
	
	// Дребезг контакторов
	_0303_05_PU01_ixKM_StatusOn_Rattling : INPUT_OUTPUT;
	_0303_05_PU02_ixKM_StatusOn_Rattling : INPUT_OUTPUT;
	_0303_05_PU03_ixKM_StatusOn_Rattling : INPUT_OUTPUT;
	_0303_05_PU04_ixKM_StatusOn_Rattling : INPUT_OUTPUT;
	_0303_05_PU05_ixKM_StatusOn_Rattling : INPUT_OUTPUT;
	_0303_05_PU01_ixKM_Frq_StatusOn_Rattling : INPUT_OUTPUT;
	_0303_05_PU02_ixKM_Frq_StatusOn_Rattling : INPUT_OUTPUT;
	_0303_05_PU03_ixKM_Frq_StatusOn_Rattling : INPUT_OUTPUT;
	_0303_05_PU04_ixKM_Frq_StatusOn_Rattling : INPUT_OUTPUT;
	_0303_05_PU05_ixKM_Frq_StatusOn_Rattling : INPUT_OUTPUT;
	_0303_05_1_ixFreq_InWork_Rattling : INPUT_OUTPUT;
	_0303_05_1_ixFreq_Manual_Rattling : INPUT_OUTPUT;
	_0303_05_1_ixFreq_Ready_Rattling : INPUT_OUTPUT;
	_0303_05_1_ixFreq_Failure_Rattling : INPUT_OUTPUT;
	_0303_05_2_ixFreq_InWork_Rattling : INPUT_OUTPUT;
	_0303_05_2_ixFreq_Manual_Rattling : INPUT_OUTPUT;
	_0303_05_2_ixFreq_Ready_Rattling : INPUT_OUTPUT;
	_0303_05_2_ixFreq_Failure_Rattling : INPUT_OUTPUT;
END_VAR

                    // Обработка команд АССУТ и сервис
_0303_05_CommandProceed(
	iiPLC_Mode:= PLC_Mode, 
	Auto_ixFrqStart:= autoCmd.Auto_ixFrqStart, 
	Auto_ixFrqChange:= autoCmd.Auto_ixFrqChange, 
	Auto_ixFrqStop:= autoCmd.Auto_ixFrqStop, 
	Auto_ixFrqEmergencyStop:= autoCmd.Auto_ixFrqEmergencyStop, 
	Auto_ixFrqReset:= autoCmd.Auto_ixFrqReset, 
	Auto_ixFrqSmoothStop:= autoCmd.Auto_ixFrqSmoothStop, 
	
	Service_ixFrqStart:= , 
	Service_ixFrqChange:= , 
	Service_ixFrqStop:= , 
	Service_ixFrqEmergencyStop:= , 
	Service_ixFrqReset:= , 
	Service_ixFrqSmoothStop:= , 
	
	Auto_iqrSetFreq:= autoCmd.Auto_iqrSetFreq, 
	Service_iqrSetFreq:= , 
	
	Auto_ixKM_PU01:= autoCmd.Auto_ixKM_PU01, 
	Auto_ixKM_PU02:= autoCmd.Auto_ixKM_PU02, 
	Auto_ixKM_PU03:= autoCmd.Auto_ixKM_PU03, 
	Auto_ixKM_PU04:= autoCmd.Auto_ixKM_PU04, 
	Auto_ixKM_PU05:= autoCmd.Auto_ixKM_PU05, 
	
	Service_ixKM_PU01:= , 
	Service_ixKM_PU02:= , 
	Service_ixKM_PU03:= , 
	Service_ixKM_PU04:= , 
	Service_ixKM_PU05:= , 
	
	qxFrqStart=> varVFD001.ixStart, 
	qxFrqChange=> varVFD001.ixChange, 
	qxFrqStop=> varVFD001.ixStop, 
	qxFrqEmergencyStop=> varVFD001.ixEmergencyStop, 
	qxFrqReset=> varVFD001.ixReset, 
	qxFrqSmoothStop=> varVFD001.ixSmoothStop, 
	qrSetFreq=> VFD001_iqrSetFreq, 
	qxKM_PU01=> ixKM_PU01, 
	qxKM_PU02=> ixKM_PU02, 
	qxKM_PU03=> ixKM_PU03, 
	qxKM_PU04=> ixKM_PU04, 
	qxKM_PU05=> ixKM_PU05);

// Статус работы контакторов ЧРП и байпас и условия обратного перехода 
CASE iIPU_Select OF
	1: 
		xKMFrqReady := NOT _0303_05_PU01_ixKM_StatusOn_Rattling.qxSignal AND NOT _0303_05_PU01_ixKM_Frq_StatusOn_Rattling.qxSignal;
		IF VFD001_rtrig_ixStart.Q OR VFD001_rtrig_ixChange.Q THEN _0303_05_PU01_qxKM_cmdOn := FALSE; END_IF;
		varVFD001.ixStarted := _0303_05_PU01_ixKM_Frq_StatusOn_Rattling.qxSignal;
	2: 		
		xKMFrqReady := NOT _0303_05_PU02_ixKM_StatusOn_Rattling.qxSignal AND NOT _0303_05_PU02_ixKM_Frq_StatusOn_Rattling.qxSignal;
		IF VFD001_rtrig_ixStart.Q OR VFD001_rtrig_ixChange.Q THEN _0303_05_PU02_qxKM_cmdOn := FALSE; END_IF;
		varVFD001.ixStarted := _0303_05_PU02_ixKM_Frq_StatusOn_Rattling.qxSignal;
	3: 
		xKMFrqReady := NOT _0303_05_PU03_ixKM_StatusOn_Rattling.qxSignal AND NOT _0303_05_PU03_ixKM_Frq_StatusOn_Rattling.qxSignal;
		IF VFD001_rtrig_ixStart.Q OR VFD001_rtrig_ixChange.Q THEN _0303_05_PU03_qxKM_cmdOn := FALSE; END_IF;
		varVFD001.ixStarted := _0303_05_PU03_ixKM_Frq_StatusOn_Rattling.qxSignal;
	4: 
		xKMFrqReady := NOT _0303_05_PU04_ixKM_StatusOn_Rattling.qxSignal AND NOT _0303_05_PU04_ixKM_Frq_StatusOn_Rattling.qxSignal;
		IF VFD001_rtrig_ixStart.Q OR VFD001_rtrig_ixChange.Q THEN _0303_05_PU04_qxKM_cmdOn := FALSE; END_IF;
		varVFD001.ixStarted := _0303_05_PU04_ixKM_Frq_StatusOn_Rattling.qxSignal;
	5: 
		xKMFrqReady := NOT _0303_05_PU05_ixKM_StatusOn_Rattling.qxSignal AND NOT _0303_05_PU05_ixKM_Frq_StatusOn_Rattling.qxSignal;
		IF VFD001_rtrig_ixStart.Q OR VFD001_rtrig_ixChange.Q THEN _0303_05_PU05_qxKM_cmdOn := FALSE; END_IF;
		varVFD001.ixStarted := _0303_05_PU05_ixKM_Frq_StatusOn_Rattling.qxSignal;
END_CASE;

VFD001(		// ЧРП ОСНОВНОЙ
	irMaxFreq:= varVFD001.irMaxFreq, 							// Максимально допустимая частота
	ixStart:= VFD001_rtrig_ixStart.Q AND xKMFrqReady, 			// Старт от rtrig при условии, что мы не получаем сигнал от контакторов байпас
	ixChange:= VFD001_rtrig_ixChange.Q,							// Переключение с байпас на ЧРП (старт без плавного пуска) 
	ixStop:= VFD001_rtrig_ixStop.Q, 							// Стоп через rtrig
	ixEmergencyStop:= varVFD001.ixEmergencyStop, 				// Аварийная остановка и отправление сигнала обратной связи ФБ
	itUpdateCycle:= varVFD001.itUpdateCycle, 					// Время обновления цикла плавного пуска/остановки в TIME 
	irUpdateCycleStep:= varVFD001.irUpdateCycleStep, 			// Шаг обновления частоты за 1 цикл
	irActualFreq:= VFD001_DebugActualFreqSim.qrActualFreq, 		// _0303_05_VFD001_MainFrq_ActualFrequency.Value - для прибора ; VFD001_DebugActualFreqSim.qrActualFreq - для симуляции		||	Получение сигнала частоты от прибора в REAL
	irActualFreqInaccuracy:= varVFD001.irActualFreqInaccuracy, 	// Максимальная допустимая погрешность для ЧРП
	ixDeviceReady:= _0303_05_1_ixFreq_Ready_Rattling.qxSignal AND NOT _0303_05_1_ixFreq_Manual_Rattling.qxSignal, // Получение сигнала о готовности от ЧРП
	ixDeviceError:= _0303_05_1_ixFreq_Failure_Rattling.qxSignal, 	// Получение сигнала об ошибке от ЧРП
	ixDeviceReserve:= FALSE,									// Статус ЧРП резерв
	ixDeviceReserveOn:= _0303_05_1_ixFreq_Failure_Rattling.qxSignal,	// Переключение работы ЧРП на резерв
	ixReset:= varVFD001.ixReset,								// Сброс всех ошибок
	ixSmoothStop := varVFD001.ixSmoothStop,						// Опция плавной остановки. TRUE - остановка происходит плавным переходом частоты от текущей до нуля, согласно шагу цикла. FALSE - остановка происходит сразу, выходная частота ФБ сбрасывается до 0.
	ixStarted := varVFD001.ixStarted,
	ixStopped := VFD001_ixStopped.Q,
	qrFreq=> , 													// SetFreqAnaloOutputSignalScale
	qxEmergencyStopStatus=> varVFD001.qxEmergencyStopStatus, 	// обратная связь ФБ
	qxStart=> , 												// по выбору насоса
	qxStartStatus=> varVFD001.qxStartStatus, 					// обратная связь ФБ
	qxStop=> , 													// по выбору насоса
	qxStopStatus=> varVFD001.qxStopStatus, 						// обратная связь ФБ
	qxErrorInvalidInaccuracy=> varVFD001.qxErrorInvalidInaccuracy, 	// обратная связь ФБ
	qxDeviceError=> varVFD001.qxDeviceError, 					// обратная связь ФБ
	qxDelayError=> varVFD001.qxDelayError,
	iqrSetFreq:= VFD001_iqrSetFreq);							// Задание частоты. При остановке сбрасывает значение до 0, после процедуры остановки возвращает прошлое значение. 

VFD002(		// ЧРП РЕЗЕРВ
	irMaxFreq:= varVFD001.irMaxFreq, 							// Максимально допустимая частота
	ixStart:= VFD001_rtrig_ixStart.Q AND xKMFrqReady, 			// Старт от rtrig при условии, что мы не получаем сигнал от контакторов байпас
	ixChange:= VFD001_rtrig_ixChange.Q,							// Переключение с байпас на ЧРП (старт без плавного пуска) 
	ixStop:= VFD001_rtrig_ixStop.Q, 							// Стоп через rtrig
	ixEmergencyStop:= varVFD002.ixEmergencyStop, 				// Аварийная остановка и отправление сигнала обратной связи ФБ
	itUpdateCycle:= varVFD001.itUpdateCycle, 					// Время обновления цикла плавного пуска/остановки в TIME 
	irUpdateCycleStep:= varVFD001.irUpdateCycleStep, 			// Шаг обновления частоты за 1 цикл
	irActualFreq:= VFD002_DebugActualFreqSim.qrActualFreq, 		// _0303_05_VFD001_MainFrq_ActualFrequency.Value - для прибора ; VFD001_DebugActualFreqSim.qrActualFreq - для симуляции		||	Получение сигнала частоты от прибора в REAL
	irActualFreqInaccuracy:= varVFD001.irActualFreqInaccuracy, 	// Максимальная допустимая погрешность для ЧРП
	ixDeviceReady:= _0303_05_2_ixFreq_Ready_Rattling.qxSignal AND NOT _0303_05_2_ixFreq_Manual_Rattling.qxSignal, // Получение сигнала о готовности от ЧРП
	ixDeviceError:= _0303_05_2_ixFreq_Failure_Rattling.qxSignal, 	// Получение сигнала об ошибке от ЧРП
	ixDeviceReserve:= TRUE,										// Статус ЧРП резерв
	ixDeviceReserveOn:= _0303_05_1_ixFreq_Failure_Rattling.qxSignal,	// Переключение работы ЧРП на резерв
	ixReset:= varVFD002.ixReset,								// Сброс всех ошибок
	ixSmoothStop := varVFD002.ixSmoothStop,						// Опция плавной остановки. TRUE - остановка происходит плавным переходом частоты от текущей до нуля, согласно шагу цикла. FALSE - остановка происходит сразу, выходная частота ФБ сбрасывается до 0.
	ixStarted := varVFD001.ixStarted,
	ixStopped := VFD001_ixStopped.Q,
	qrFreq=> , 													// SetFreqAnaloOutputSignalScale
	qxEmergencyStopStatus=> varVFD002.qxEmergencyStopStatus, 	// обратная связь ФБ
	qxStart=> , 												// по выбору насоса
	qxStartStatus=> varVFD002.qxStartStatus, 					// обратная связь ФБ
	qxStop=> , 													// по выбору насоса
	qxStopStatus=> varVFD002.qxStopStatus, 						// обратная связь ФБ
	qxErrorInvalidInaccuracy=> varVFD002.qxErrorInvalidInaccuracy, 	// обратная связь ФБ
	qxDeviceError=> varVFD002.qxDeviceError, 					// обратная связь ФБ
	qxDelayError=> ,
	iqrSetFreq:= VFD001_iqrSetFreq);							// Задание частоты. При остановке сбрасывает значение до 0, после процедуры остановки возвращает прошлое значение. 
	
VFD001_rtrig_ixStop(CLK:= varVFD001.ixStop, Q=> );				// Стоп работы VFD001
VFD001_rtrig_ixChange(CLK:= varVFD001.ixChange, Q=> );			// Старт работы VFD001 (без плавного пуска)
VFD001_rtrig_ixStart(CLK:= varVFD001.ixStart, Q=> );			// Старт работы VFD001

xPuKmFrqWorked := 
	_0303_05_PU01_ixKM_Frq_StatusOn_Rattling.qxSignal
	OR _0303_05_PU02_ixKM_Frq_StatusOn_Rattling.qxSignal
	OR _0303_05_PU03_ixKM_Frq_StatusOn_Rattling.qxSignal
	OR _0303_05_PU04_ixKM_Frq_StatusOn_Rattling.qxSignal
	OR _0303_05_PU05_ixKM_Frq_StatusOn_Rattling.qxSignal;

VFD001_ixStopped(CLK:= xPuKmFrqWorked, Q=> );
	
//	=====	ОТЛАДКА		====

// Симуляция получения сигнала частоты от прибора
VFD001_DebugActualFreqSim(
	irOrderFreq:= VFD001.qrFreq, 
	irInac:= 0.1, 
	itDelay:= T#100MS, 
	ixReverseInac:= , 
	qrActualFreq=> VFD001.irActualFreq);
	
VFD002_DebugActualFreqSim(
	irOrderFreq:= VFD002.qrFreq, 
	irInac:= 0.1, 
	itDelay:= T#100MS, 
	ixReverseInac:= , 
	qrActualFreq=> VFD002.irActualFreq);

// 	========================

// Конвертация REAL выходного сигнала ФБ VFD001-2.qrFreq в UINT сигнал 0..1000 для модуля аналогового выхода, настроенного на 4..20мА
SetFreqAnaloOutputSignalScale(
	irSetFrequencyHz:= VFD001.qrFreq, 
	irSetFrequencyHzMax:= varVFD001.irMaxFreq, 
	qIScaledValue=> );
_0303_05_VFD001_qIMainFrq_SetFrq := SetFreqAnaloOutputSignalScale.qIScaledValue;
_0303_05_VFD002_qIReserveFrq_SetFrq := SetFreqAnaloOutputSignalScale.qIScaledValue;

// Условия включения контактора ЧРП основной и резерв
IF ix1KM8_qxOn THEN _0303_05_1KM8_qxOn := TRUE; 
ELSIF ix1KM8_qxOff THEN _0303_05_1KM8_qxOn := FALSE; END_IF;

IF ix2KM8_qxOn THEN _0303_05_2KM8_qxOn := TRUE;
ELSIF ix2KM8_qxOff THEN _0303_05_2KM8_qxOn := FALSE; END_IF;


// Насос PU1 включение через ЧРП и условия переключения на байпас
RS_0303_05_PU01_qxKM_Frq_cmdOn(
	SET:= (VFD001.qxStart AND NOT VFD001.ixDeviceReserveOn) OR (VFD002.qxStart AND VFD001.ixDeviceReserveOn) AND iIPU_Select = 1, 
	RESET1:= (VFD001.qxStop OR (varVFD001.ixEmergencyStop OR varVFD002.ixEmergencyStop) OR ixKM_PU01) AND iIPU_Select = 1, 
	Q1=>_0303_05_PU01_qxKM_Frq_cmdOn );

// Насос PU2 включение через ЧРП и условия переключения на байпас
RS_0303_05_PU02_qxKM_Frq_cmdOn(
	SET:= (VFD001.qxStart AND NOT VFD001.ixDeviceReserveOn) OR (VFD002.qxStart AND VFD001.ixDeviceReserveOn) AND iIPU_Select = 2, 
	RESET1:= (VFD001.qxStop OR (varVFD001.ixEmergencyStop OR varVFD002.ixEmergencyStop) OR ixKM_PU01) AND iIPU_Select = 2, 
	Q1=>_0303_05_PU02_qxKM_Frq_cmdOn );
	
// Насос PU3 включение через ЧРП и условия переключения на байпас
RS_0303_05_PU03_qxKM_Frq_cmdOn(
	SET:= (VFD001.qxStart AND NOT VFD001.ixDeviceReserveOn) OR (VFD002.qxStart AND VFD001.ixDeviceReserveOn) AND iIPU_Select = 3, 
	RESET1:= (VFD001.qxStop OR (varVFD001.ixEmergencyStop OR varVFD002.ixEmergencyStop) OR ixKM_PU01) AND iIPU_Select = 3, 
	Q1=>_0303_05_PU03_qxKM_Frq_cmdOn );
	
// Насос PU4 включение через ЧРП и условия переключения на байпас
RS_0303_05_PU04_qxKM_Frq_cmdOn(
	SET:= (VFD001.qxStart AND NOT VFD001.ixDeviceReserveOn) OR (VFD002.qxStart AND VFD001.ixDeviceReserveOn) AND iIPU_Select = 4, 
	RESET1:= (VFD001.qxStop OR (varVFD001.ixEmergencyStop OR varVFD002.ixEmergencyStop) OR ixKM_PU01) AND iIPU_Select = 4, 
	Q1=>_0303_05_PU04_qxKM_Frq_cmdOn );
	
// Насос PU5 включение через ЧРП и условия переключения на байпас
RS_0303_05_PU05_qxKM_Frq_cmdOn(
	SET:= (VFD001.qxStart AND NOT VFD001.ixDeviceReserveOn) OR (VFD002.qxStart AND VFD001.ixDeviceReserveOn) AND iIPU_Select = 5, 
	RESET1:= (VFD001.qxStop OR (varVFD001.ixEmergencyStop OR varVFD002.ixEmergencyStop) OR ixKM_PU01) AND iIPU_Select = 5, 
	Q1=>_0303_05_PU05_qxKM_Frq_cmdOn );

// Переключение с ЧРП на байпас
IF ixKM_PU01 AND NOT _0303_05_PU01_ixKM_Frq_StatusOn_Rattling.qxSignal AND iIPU_Select = 1 THEN _0303_05_PU01_qxKM_cmdOn := TRUE; varVFD001.ixStop := TRUE; iIPU_Select := 0; END_IF;
IF ixKM_PU02 AND NOT _0303_05_PU02_ixKM_Frq_StatusOn_Rattling.qxSignal AND iIPU_Select = 2 THEN _0303_05_PU02_qxKM_cmdOn := TRUE; varVFD001.ixStop := TRUE; iIPU_Select := 0; END_IF;
IF ixKM_PU03 AND NOT _0303_05_PU03_ixKM_Frq_StatusOn_Rattling.qxSignal AND iIPU_Select = 3 THEN _0303_05_PU03_qxKM_cmdOn := TRUE; varVFD001.ixStop := TRUE; iIPU_Select := 0; END_IF;
IF ixKM_PU04 AND NOT _0303_05_PU04_ixKM_Frq_StatusOn_Rattling.qxSignal AND iIPU_Select = 4 THEN _0303_05_PU04_qxKM_cmdOn := TRUE; varVFD001.ixStop := TRUE; iIPU_Select := 0; END_IF;
IF ixKM_PU05 AND NOT _0303_05_PU05_ixKM_Frq_StatusOn_Rattling.qxSignal AND iIPU_Select = 5 THEN _0303_05_PU05_qxKM_cmdOn := TRUE; varVFD001.ixStop := TRUE; iIPU_Select := 0; END_IF;

// Работа затвора _0303_05_BY01
_0303_05_BY01(
	time_error_long_time_without_status:= , // inactive
	ixready:= _0303_05_BY01_ixShutter_StatusReady_FB.qxSignal, 
	ixerror:= _0303_05_BY01_ixShutter_StatusError_FB.qxSignal, 
	ixopen:= _0303_05_BY01_Contactor_PosOpen_FB.qxSignal, 
	ixclose:= _0303_05_BY01_Contactor_PosClosed_FB.qxSignal, 
	ixreset:= _0303_05_BY01_ixreset, 
	ixopened_status:= _0303_05_BY01_ixShutter_PosOpen_FB.qxSignal, 
	ixclosed_status:= _0303_05_BY01_ixShutter_PosClosed_FB.qxSignal, 
	qxopen=> _0303_05_BY01_qxShutter_Open, 
	qxclose=> _0303_05_BY01_qxShutter_Close, 
	qxerror_from_device=> , // обр. связь
	qxopened=> , 			// обр. связь
	qxclosed=> , 			// обр. связь
	qxclose_process=> , 	// обр. связь
	qxopen_process=> );		// обр. связь
	
_0303_05_BY01_Contactor_PosOpen_FB(
	ixSignal:= _0303_05_BY01_ixKM_PosOpen, 
	itInputTime:= inputOutput_ButtonInputTime, 
	itRattling_count_reset:= , 
	ixResetAlarm:= , // обр. связь
	qxSignal=> , // _0303_05_BY01
	qxRattlingAlarm=> ); // обр. связь
	
_0303_05_BY01_Contactor_PosClosed_FB(
	ixSignal:= _0303_05_BY01_ixKM_PosClosed, 
	itInputTime:= inputOutput_ButtonInputTime, 
	itRattling_count_reset:= , 
	ixResetAlarm:= , // обр. связь
	qxSignal=> , // _0303_05_BY01
	qxRattlingAlarm=> ); // обр. связь
	
_0303_05_BY01_ixShutter_StatusReady_FB(
	ixSignal:= _0303_05_BY01_ixShutter_StatusReady, 
	itInputTime:= inputOutput_ButtonInputTime, 
	itRattling_count_reset:= , 
	ixResetAlarm:= , 
	qxSignal=> , // _0303_05_BY01
	qxRattlingAlarm=> );
	
_0303_05_BY01_ixShutter_StatusError_FB(
	ixSignal:= _0303_05_BY01_ixShutter_StatusError, 
	itInputTime:= inputOutput_ButtonInputTime, 
	itRattling_count_reset:= , 
	ixResetAlarm:= , 
	qxSignal=> , // _0303_05_BY01
	qxRattlingAlarm=> );
	
_0303_05_BY01_ixShutter_PosOpen_FB(
	ixSignal:= _0303_05_BY01_ixShutter_PosOpen, 
	itInputTime:= inputOutput_ButtonInputTime, 
	itRattling_count_reset:= , 
	ixResetAlarm:= , 
	qxSignal=> , // _0303_05_BY01
	qxRattlingAlarm=> );
	
_0303_05_BY01_ixShutter_PosClosed_FB(
	ixSignal:= _0303_05_BY01_ixShutter_PosClosed, 
	itInputTime:= inputOutput_ButtonInputTime, 
	itRattling_count_reset:= , 
	ixResetAlarm:= , 
	qxSignal=> , // _0303_05_BY01
	qxRattlingAlarm=> );
	
// ДРЕБЕЗГ КОНТАКТОРОВ

// Контакторы статуса насосов (байпас)
_0303_05_PU01_ixKM_StatusOn_Rattling(
	ixSignal:= _0303_05_PU01_ixKM_StatusOn, 
	itInputTime:= inputOutput_ButtonInputTime, 
	itRattling_count_reset:= , 
	ixResetAlarm:= , 
	qxSignal=> , 
	qxRattlingAlarm=> );

_0303_05_PU02_ixKM_StatusOn_Rattling(
	ixSignal:= _0303_05_PU02_ixKM_StatusOn, 
	itInputTime:= inputOutput_ButtonInputTime, 
	itRattling_count_reset:= , 
	ixResetAlarm:= , 
	qxSignal=> , 
	qxRattlingAlarm=> );
	
_0303_05_PU03_ixKM_StatusOn_Rattling(
	ixSignal:= _0303_05_PU03_ixKM_StatusOn, 
	itInputTime:= inputOutput_ButtonInputTime, 
	itRattling_count_reset:= , 
	ixResetAlarm:= , 
	qxSignal=> , 
	qxRattlingAlarm=> );

_0303_05_PU04_ixKM_StatusOn_Rattling(
	ixSignal:= _0303_05_PU04_ixKM_StatusOn, 
	itInputTime:= inputOutput_ButtonInputTime, 
	itRattling_count_reset:= , 
	ixResetAlarm:= , 
	qxSignal=> , 
	qxRattlingAlarm=> );

_0303_05_PU05_ixKM_StatusOn_Rattling(
	ixSignal:= _0303_05_PU05_ixKM_StatusOn, 
	itInputTime:= inputOutput_ButtonInputTime, 
	itRattling_count_reset:= , 
	ixResetAlarm:= , 
	qxSignal=> , 
	qxRattlingAlarm=> );

// Контакторы статус ЧРП ОСНОВНОЙ
_0303_05_1_ixFreq_InWork_Rattling(
	ixSignal:= _0303_05_1_ixVFD_InWork, 
	itInputTime:= inputOutput_ButtonInputTime, 
	itRattling_count_reset:= , 
	ixResetAlarm:= , 
	qxSignal=> , 
	qxRattlingAlarm=> );

_0303_05_1_ixFreq_Manual_Rattling(
	ixSignal:= _0303_05_1_ixVFD_Manual, 
	itInputTime:= inputOutput_ButtonInputTime, 
	itRattling_count_reset:= , 
	ixResetAlarm:= , 
	qxSignal=> , 
	qxRattlingAlarm=> );
	
_0303_05_1_ixFreq_Ready_Rattling(
	ixSignal:= _0303_05_1_ixVFD_Ready, 
	itInputTime:= inputOutput_ButtonInputTime, 
	itRattling_count_reset:= , 
	ixResetAlarm:= , 
	qxSignal=> , 
	qxRattlingAlarm=> );

_0303_05_1_ixFreq_Failure_Rattling(
	ixSignal:= _0303_05_1_ixVFD_Failure, 
	itInputTime:= inputOutput_ButtonInputTime, 
	itRattling_count_reset:= , 
	ixResetAlarm:= , 
	qxSignal=> , 
	qxRattlingAlarm=> );

// Контакторы статус ЧРП РЕЗЕРВ
_0303_05_2_ixFreq_InWork_Rattling(
	ixSignal:= _0303_05_2_ixVFD_InWork, 
	itInputTime:= inputOutput_ButtonInputTime, 
	itRattling_count_reset:= , 
	ixResetAlarm:= , 
	qxSignal=> , 
	qxRattlingAlarm=> );

_0303_05_2_ixFreq_Manual_Rattling(
	ixSignal:= _0303_05_2_ixVFD_Manual, 
	itInputTime:= inputOutput_ButtonInputTime, 
	itRattling_count_reset:= , 
	ixResetAlarm:= , 
	qxSignal=> , 
	qxRattlingAlarm=> );
	
_0303_05_2_ixFreq_Ready_Rattling(
	ixSignal:= _0303_05_2_ixVFD_Ready, 
	itInputTime:= inputOutput_ButtonInputTime, 
	itRattling_count_reset:= , 
	ixResetAlarm:= , 
	qxSignal=> , 
	qxRattlingAlarm=> );

_0303_05_2_ixFreq_Failure_Rattling(
	ixSignal:= _0303_05_2_ixVFD_Failure, 
	itInputTime:= inputOutput_ButtonInputTime, 
	itRattling_count_reset:= , 
	ixResetAlarm:= , 
	qxSignal=> , 
	qxRattlingAlarm=> );

// Контакторы насосов (ЧРП)
_0303_05_PU01_ixKM_Frq_StatusOn_Rattling(
	ixSignal:= _0303_05_PU01_ixKM_VFD_StatusOn, 
	itInputTime:= inputOutput_ButtonInputTime, 
	itRattling_count_reset:= , 
	ixResetAlarm:= , 
	qxSignal=> , 
	qxRattlingAlarm=> );
	
_0303_05_PU02_ixKM_Frq_StatusOn_Rattling(
	ixSignal:= _0303_05_PU02_ixKM_VFD_StatusOn, 
	itInputTime:= inputOutput_ButtonInputTime, 
	itRattling_count_reset:= , 
	ixResetAlarm:= , 
	qxSignal=> , 
	qxRattlingAlarm=> );
	
_0303_05_PU03_ixKM_Frq_StatusOn_Rattling(
	ixSignal:= _0303_05_PU03_ixKM_VFD_StatusOn, 
	itInputTime:= inputOutput_ButtonInputTime, 
	itRattling_count_reset:= , 
	ixResetAlarm:= , 
	qxSignal=> , 
	qxRattlingAlarm=> );
	
_0303_05_PU04_ixKM_Frq_StatusOn_Rattling(
	ixSignal:= _0303_05_PU04_ixKM_VFD_StatusOn, 
	itInputTime:= inputOutput_ButtonInputTime, 
	itRattling_count_reset:= , 
	ixResetAlarm:= , 
	qxSignal=> , 
	qxRattlingAlarm=> );
	
_0303_05_PU05_ixKM_Frq_StatusOn_Rattling(
	ixSignal:= _0303_05_PU05_ixKM_VFD_StatusOn, 
	itInputTime:= inputOutput_ButtonInputTime, 
	itRattling_count_reset:= , 
	ixResetAlarm:= , 
	qxSignal=> , 
	qxRattlingAlarm=> );
                  
END_PROGRAM

FUNCTION_BLOCK FB_Asignal_FreqConvertation
VAR_INPUT
    irSetFrequencyHz : REAL; // частота в Гц
	irSetFrequencyHzMax : REAL; // максимальная частота
END_VAR

VAR_OUTPUT
    qIScaledValue : UINT; // масштабированное значение для аналогово выхода (0 .. 1000)
END_VAR

VAR
    TempValue : REAL;
END_VAR

                    // Вход: SetFrequencyHz : REAL (0.0 .. 50.0)
// Выход: ScaledValue : UINT (0 .. 1000)

// Масштабирование: (SetFrequencyHz / 50.0) * 1000
TempValue := (irSetFrequencyHz / irSetFrequencyHzMax) * 1000.0;

// Обрезка границ
IF TempValue < 0.0 THEN
    qIScaledValue := 0;
ELSIF TempValue > 1000.0 THEN
    qIScaledValue := 1000;
ELSE
	qIScaledValue := REAL_TO_UINT(TempValue);
END_IF;

                  
END_FUNCTION_BLOCK

FUNCTION_BLOCK FB_CommandProceed
VAR_INPUT
	iiPLC_Mode : INT; // 0 – «Авто», 1 – «Обрыв связи», 2 – «Местный-Сервис»
	
	Auto_ixFrqStart : BOOL;
	Auto_ixFrqChange : BOOL;
	Auto_ixFrqStop : BOOL;
	Auto_ixFrqEmergencyStop : BOOL;
	Auto_ixFrqReset : BOOL;
	Auto_ixFrqSmoothStop : BOOL;
	
	Service_ixFrqStart : BOOL;
	Service_ixFrqChange : BOOL;
	Service_ixFrqStop : BOOL;
	Service_ixFrqEmergencyStop : BOOL;
	Service_ixFrqReset : BOOL;
	Service_ixFrqSmoothStop : BOOL;
	
	Auto_iqrSetFreq : REAL;
	Service_iqrSetFreq : REAL;
	
	Auto_ixKM_PU01 : BOOL;
	Auto_ixKM_PU02 : BOOL;
	Auto_ixKM_PU03 : BOOL;
	Auto_ixKM_PU04 : BOOL;
	Auto_ixKM_PU05 : BOOL;
	
	Service_ixKM_PU01 : BOOL;
	Service_ixKM_PU02 : BOOL;
	Service_ixKM_PU03 : BOOL;
	Service_ixKM_PU04 : BOOL;
	Service_ixKM_PU05: BOOL;
	
END_VAR
VAR_OUTPUT
	qxFrqStart : BOOL;
	qxFrqChange : BOOL;
	qxFrqStop : BOOL;
	qxFrqEmergencyStop : BOOL;
	qxFrqReset : BOOL;
	qxFrqSmoothStop : BOOL;
	
	qrSetFreq : REAL;
	
	qxKM_PU01 : BOOL;
	qxKM_PU02 : BOOL;
	qxKM_PU03 : BOOL;
	qxKM_PU04 : BOOL;
	qxKM_PU05 : BOOL;
END_VAR
VAR
END_VAR

                    IF iiPLC_Mode = 0 THEN
	qxFrqStart := Auto_ixFrqStart;
	qxFrqChange := Auto_ixFrqChange;
	qxFrqStop := Auto_ixFrqStop;
	qxFrqEmergencyStop := Auto_ixFrqEmergencyStop;
	qxFrqReset := Auto_ixFrqReset;
	qxFrqSmoothStop := Auto_ixFrqSmoothStop;
	
	qrSetFreq := Auto_iqrSetFreq;
	
	qxKM_PU01 := Auto_ixKM_PU01;
	qxKM_PU02 := Auto_ixKM_PU02;
	qxKM_PU03 := Auto_ixKM_PU03;
	qxKM_PU04 := Auto_ixKM_PU04;
	qxKM_PU05 := Auto_ixKM_PU05;
END_IF;

IF iiPLC_Mode = 2 THEN
	qxFrqStart := Service_ixFrqStart;
	qxFrqChange := Service_ixFrqChange;
	qxFrqStop := Service_ixFrqStop;
	qxFrqEmergencyStop := Service_ixFrqEmergencyStop;
	qxFrqReset := Service_ixFrqReset;
	qxFrqSmoothStop := Service_ixFrqSmoothStop;
	
	qrSetFreq := Service_iqrSetFreq;
	
	qxKM_PU01 := Service_ixKM_PU01;
	qxKM_PU02 := Service_ixKM_PU02;
	qxKM_PU03 := Service_ixKM_PU03;
	qxKM_PU04 := Service_ixKM_PU04;
	qxKM_PU05 := Service_ixKM_PU05;
END_IF;
                  
END_FUNCTION_BLOCK

FUNCTION_BLOCK FB_TEST_A_SIGNAL_SCALE
VAR_INPUT
	irSignal : REAL; 			// Вход аналогового сигнала
	irSignalSim : REAL; 		// Вход аналогового сигнала (симулятор)
	irSignalDownLimit : REAL; 	// Нижний предел сигнала
	irSignalUpLimit : REAL; 	// Верхний предел сигнала
	
	irValueDownLimit : REAL; 	// Нижний предел масштабированной единицы
	irValueUpLimit : REAL; 		// Верхий предел масштабированной единицы
	
	irHSignal : REAL; 			// Верхний предупредительный сигнал
	irHHSignal : REAL; 			// Верхний аварийный сигнал
	irLSignal : REAL; 			// Нижний предупредительный сигнал
	irLLSignal : REAL; 			// Верхний предупредительный сигнал
	
	ixReset : BOOL; 			// Ресет ошибок
	ixDeviceOn : BOOL; 			// Датчик работает
	
	ixSimulation : BOOL;		// Режим симуляции сигнала
	ixAlarmMode : BOOL; 		// Режим отображения L LL H HH сигналов
END_VAR
VAR_OUTPUT
	qrSignal : REAL; 			// Выходной масштабированный сигнал
	qxMaxSignal : BOOL;			// Достижение минимального сигнала
	qxMinSignal : BOOL; 		// Достижение максимального сигнала
	qxErrorMin : BOOL; 			// Ошибка: сигнал меньше, чем минимально допустимый
	qxErrorMax : BOOL; 			// Ошибка: сигнал больше, чем максимально допустимый
	qxHSignal : BOOL; 			// Достижение верхнего предупредительного сигнала
	qxHHSignal : BOOL; 			// Достижение верхнего аварийного сигнала 
	qxLSignal : BOOL;			// Достижение нижнего предупредительного сигнала
	qxLLSignal : BOOL;			// Достижение нихнего аварийного сигнала
END_VAR
VAR
	rtrig_ixReset : R_TRIG;
END_VAR

                    rtrig_ixReset(CLK:= ixReset, Q=> );
ResetError(rtrig_ixReset.Q);
ResetAlarm(rtrig_ixReset.Q);

IF NOT ixSimulation AND ixDeviceOn THEN 
	qrSignal := ScaleSignal(irSignal);
	GetFeedback(); 
END_IF;

IF ixSimulation AND ixDeviceOn THEN
	qrSignal := ScaleSignal(irSignalSim); 
	GetFeedback();
END_IF;

IF ixAlarmMode THEN 
	AlarmMode(); 
	ResetAlarm(rtrig_ixReset.Q); 
END_IF;
                  

METHOD ScaleSignal : REAL
VAR_INPUT
	A_Signal : REAL;
END_VAR
                          ScaleSignal := ((A_Signal - irSignalDownLimit) * (irValueUpLimit - irValueDownLimit)) / (irSignalUpLimit - irSignalDownLimit) + irValueDownLimit;
                        
END_METHOD

METHOD ResetError : BOOL
VAR_INPUT
	xResetSignal : BOOL;
END_VAR
                          IF xResetSignal THEN
	qxMaxSignal := FALSE;
	qxMinSignal := FALSE;
	qxErrorMax := FALSE;
	qxErrorMin := FALSE;
END_IF;
                        
END_METHOD

METHOD GetFeedback : BOOL
VAR_INPUT
END_VAR
VAR
// 	rtrig_qxMinSignal : R_TRIG;
// 	rtrig_qxMaxSignal : R_TRIG;
	
	rtrig_qxErrorMin : R_TRIG;
	rtrig_qxErrorMax : R_TRIG;
END_VAR
                          // rtrig_qxMinSignal(CLK:= qrSignal = irValueDownLimit, Q=> );
// rtrig_qxMaxSignal(CLK:= qrSignal = irValueUpLimit, Q=> );
rtrig_qxErrorMin(CLK:= qrSignal < irValueDownLimit, Q=> );
rtrig_qxErrorMax(CLK:= qrSignal > irValueDownLimit, Q=> );


qxMinSignal := qrSignal = irValueDownLimit;
qxMaxSignal := qrSignal = irValueUpLimit;

IF rtrig_qxErrorMin.Q THEN qxErrorMin := TRUE; END_IF;
IF rtrig_qxErrorMax.Q THEN qxErrorMax := TRUE; END_IF;
                        
END_METHOD

METHOD GetAlarmL : BOOL
VAR_INPUT
	rLlimit : REAL;
END_VAR
                          GetAlarmL := rLlimit > qrSignal;
                        
END_METHOD

METHOD AlarmMode : BOOL
VAR_INPUT
END_VAR
                          IF ixAlarmMode THEN
	IF GetAlarmH(irHSignal) THEN qxHSignal := TRUE; END_IF;	// Верхний предупредительный
	IF GetAlarmH(irHHSignal) THEN qxHHSignal := TRUE; END_IF;	// Верхний аварийный
	IF GetAlarmL(irLSignal) THEN qxLSignal := TRUE; END_IF; 	// Нижний предупредительный
	IF GetAlarmL(irLSignal) THEN qxLLSignal := TRUE; END_IF;	// Нижний аварийный
END_IF;
                        
END_METHOD

METHOD GetAlarmH : BOOL
VAR_INPUT
	rHLimit : REAL;
END_VAR
                          GetAlarmH := rHLimit < qrSignal;
                        
END_METHOD

METHOD ResetAlarm : BOOL
VAR_INPUT
	xResetSignal : BOOL;
END_VAR
                          IF xResetSignal THEN
	qxHSignal := FALSE;
	qxHHSignal := FALSE;
	qxLSignal := FALSE;
	qxLLSignal := FALSE;
END_IF;
                        
END_METHOD
END_FUNCTION_BLOCK

FUNCTION_BLOCK FB_Shutter_Test IMPLEMENTS IShutterCommands, IShutterFeedback
VAR_INPUT
	ixOpenCmd : BOOL;	// Команда открыть
	ixCloseCmd : BOOL;	// Команда закрыть
	ixStopCmd : BOOL;	// Команда остановить
	ixResetCmd : BOOL;	// Сброс всех ошибок
	
	ixReadyStatus : BOOL;	// Состояние - готов.
	ixErrorCommonStatus : BOOL;	// Авария - обобщённая
	ixManualStatus : BOOL;	// ЗРА в местном управлении
	ixOpenStatus : BOOL;	// Статус - открыт
	ixClosedStatus : BOOL; 	// Статус - закрыт
END_VAR
VAR_OUTPUT
	qxOpen : BOOL;		// Открытие затвора
	qxClose : BOOL;		// Закрытие затвора
	
	qxErrorCommonStatus : BOOL; 	// Транзит сигнала ошибки ЗРА
	qxManualStatus : BOOL;			// Транзит сигнала ручного управления
	qxStoppedStatus : BOOL;			// Сигнал ЗРА остановлен
	qxOpenProcessStatus : BOOL;		// Процесс открытия затвора
	qxCloseProcessStatus : BOOL;	// Процесс закрытия затвора
	qxOpenStatus : BOOL;	// Статус - открыт
	qxClosedStatus : BOOL; 	// Статус - закрыт
END_VAR
VAR
END_VAR

                    UpdateFeedbackProcess();
CloseOpenProcess();
                  

METHOD UpdateFeedbackProcess : BOOL
VAR_INPUT
END_VAR
VAR
	ftrig_qxOpenProcessStatus : F_TRIG;
	ftrig_qxCloseProcessStatus : F_TRIG;
END_VAR
                          ftrig_qxOpenProcessStatus(CLK:= qxOpen, Q=> );
ftrig_qxCloseProcessStatus(CLK:= qxClose, Q=> );

IF ftrig_qxOpenProcessStatus.Q THEN qxOpenProcessStatus := FALSE; END_IF;
IF ftrig_qxCloseProcessStatus.Q THEN qxCloseProcessStatus := FALSE; END_IF;

qxOpenStatus := GetStatusOpen();
qxClosedStatus := GetStatusClosed();

qxManualStatus := GetStatusManual();

qxErrorCommonStatus := GetStatusCommonError();

                        
END_METHOD

METHOD OpenCloseProcessStatus : BOOL
VAR_INPUT
END_VAR
                          OpenCloseProcessStatus := qxOpen OR qxClose;
                        
END_METHOD

METHOD CloseOpenProcess : BOOL
VAR_INPUT
END_VAR
VAR
	xOpen : BOOL;
	xClose : BOOL;
	
	rtrig_ixOpenCmd : R_TRIG;
	rtrig_ixCloseCmd : R_TRIG;
	rtrig_ixStopCmd : R_TRIG;
	rtrig_ixResetCmd : R_TRIG;
	
	rtrig_ixOpenStatus : R_TRIG;
	rtrig_ixClosedStatus : R_TRIG;
	
END_VAR
                          rtrig_ixOpenCmd(CLK:= ixOpenCmd, Q=> );
rtrig_ixCloseCmd(CLK:= ixCloseCmd, Q=> );
rtrig_ixStopCmd(CLK:= ixStopCmd, Q=> );
rtrig_ixResetCmd(CLK:= ixResetCmd, Q=> );

rtrig_ixOpenStatus(CLK:= ixOpenStatus, Q=> );
rtrig_ixClosedStatus(CLK:= ixClosedStatus, Q=> );

IF NOT GetStatusManual() THEN
	IF rtrig_ixOpenCmd.Q AND GetStatusReady() AND NOT GetStatusOpen() THEN
		cmdOpen(TRUE);
	END_IF;
	
	IF rtrig_ixCloseCmd.Q AND GetStatusReady() AND NOT GetStatusClosed() THEN
		cmdClose(TRUE);
	END_IF;
	
	IF OpenCloseProcessStatus() AND GetStatusOpen() THEN
		cmdOpen(FALSE);
	END_IF;
	
	IF OpenCloseProcessStatus() AND GetStatusClosed() THEN
		cmdClose(FALSE);
	END_IF;
	
	IF rtrig_ixStopCmd.Q THEN
		cmdStop(TRUE);
	END_IF;
	
	IF rtrig_ixResetCmd.Q THEN cmdReset(); END_IF;

END_IF;
                        
END_METHOD

{warning 'добавить реализацию метода'}
METHOD cmdClose : BOOL
VAR_INPUT
	xClose : BOOL;
END_VAR
VAR
END_VAR
                          IF xClose THEN
	qxClose := TRUE;
	qxCloseProcessStatus := TRUE;
	qxStoppedStatus := FALSE;
ELSIF NOT xClose THEN
	qxClose := FALSE;
	qxCloseProcessStatus := FALSE;
END_IF;
                        
END_METHOD

{warning 'добавить реализацию метода'}
METHOD cmdOpen : BOOL
VAR_INPUT
	xOpen	: BOOL;
END_VAR
                          IF xOpen THEN
	qxOpen := TRUE;
	qxOpenProcessStatus := TRUE;
	qxStoppedStatus := FALSE;
ELSIF NOT xOpen THEN
	qxOpen := FALSE;
	qxOpenProcessStatus := FALSE;
END_IF;
                        
END_METHOD

{warning 'добавить реализацию метода'}
METHOD cmdReset : BOOL
VAR_INPUT
END_VAR
                          qxErrorCommonStatus := FALSE;

  
                        
END_METHOD

{warning 'добавить реализацию метода'}
METHOD cmdStop : BOOL
VAR_INPUT
	xStop	: BOOL;
END_VAR
                          IF xStop THEN
	cmdClose(FALSE);
	cmdOpen(FALSE);
	qxStoppedStatus := TRUE;
END_IF;
                        
END_METHOD

{warning 'добавить реализацию метода'}
METHOD GetStatusClosed : BOOL
VAR_INPUT
END_VAR
                          GetStatusClosed := ixClosedStatus;
                        
END_METHOD

{warning 'добавить реализацию метода'}
METHOD GetStatusCommonError : BOOL
VAR_INPUT
END_VAR
                          GetStatusCommonError := ixErrorCommonStatus;
                        
END_METHOD

{warning 'добавить реализацию метода'}
METHOD GetStatusManual : BOOL
VAR_INPUT
END_VAR
                          GetStatusManual := ixManualStatus;
                        
END_METHOD

{warning 'добавить реализацию метода'}
METHOD GetStatusOpen : BOOL
VAR_INPUT
END_VAR
                          GetStatusOpen := ixOpenStatus;
                        
END_METHOD

{warning 'добавить реализацию метода'}
METHOD GetStatusReady : BOOL
VAR_INPUT
END_VAR
                          GetStatusReady := ixReadyStatus;
                        
END_METHOD
END_FUNCTION_BLOCK

FUNCTION_BLOCK FB_VFD_CTRL
VAR_INPUT
//	Конфигурация
	irMaxFreq : REAL; 			// Максимальное задание частоты
	itUpdateCycle : TIME; 		// Время обновления цикла плавного пуска/остановки в TIME 
	irUpdateCycleStep : REAL; 	// Шаг обновления частоты за 1 цикл
	irActualFreqInaccuracy : REAL;	// Максимальная допустимая погрешность для ЧРП
	ixSmoothStop : BOOL;		// Режим плавной остановки
	itStartStopDelay : TIME;	// Время задержки сигнала старт и стоп до его отключения и выхода ошибки долгого ожидания отклика механизма
	
//	Команды
	ixStart : BOOL;				// Запуск
	ixFastStart : BOOL;			// Запуск без плавного задания частоты
	ixStop : BOOL;				// Остановка
	ixEmergencyStop : BOOL;		// Аварийная остановка (сброс с выходным статусом)
	ixReset : BOOL;				// Сброс ошибок ФБ
	
//	Получение сигналов
	ixStarted : BOOL;			// Получение сигнала о старте механизма
	ixStopped : BOOL;			// Получение сигнала о стопе механизма
	ixDeviceError : BOOL;		// Ошибка исполнительного механизма
	ixDeviceReady : BOOL;		// Готовность исполнительного механизма
	irActualFreq : REAL;		// Показания текущей частоты устройства
END_VAR
VAR_OUTPUT
// 	Основное
	qrFreq : REAL;				// Задание частоты на выход
	qxStart : BOOL;				// Запуск исполнительного механизма
	qxStop : BOOL;				// Остановка исполнительного механизма

// Обратная связь
	qxStartStatus : BOOL;						// Статус запуска
	qxStopStatus : BOOL;						// Статус остановки
	qxEmergencyStopStatus : BOOL;				// Статус аварийной остановки
	qxErrorInvalidInaccuracy : BOOL;			// Ошибка большой погрешности
	qxErrorDevice : BOOL;						// Ошибка исполнительного механизма (транзит через блок)
	qxDelayError : BOOL;						// Ошибка долгого ожидания обратной связи механизма после выполнения
END_VAR
VAR_IN_OUT
// Основное
	iqrSetFreq : REAL;			// Задание частоты на вход
END_VAR
VAR
	blink_updateCycle : BLINK;
	xWorkProcess : BOOL;
	xPossibleInac : BOOL;
	xErrorFixation : BOOL;
	ton_stopWorkProcess : TON;
	ton_StopDisable : TON;
	ton_StartDisable : TON;
	reserve_iqrSetFreq : REAL;
	
	rtrig_updateCycle : R_TRIG;
	rtrig_ixStart : R_TRIG;
	rtrig_ixFastStart : R_TRIG;
	rtrig_ixStop : R_TRIG;
	rtrig_ixEmergencyStop : R_TRIG;
	rtrig_ixReset : R_TRIG;
	rtrig_ixStarted : R_TRIG;
	rtrig_ixStopped : R_TRIG;
	ftrig_StopWorkProcess : F_TRIG;
END_VAR

                    rtrig_ixStart(CLK:= ixStart, Q=> );
rtrig_ixFastStart(CLK:= ixFastStart, Q=> );
rtrig_ixStop(CLK:= ixStop, Q=> );
ftrig_StopWorkProcess(CLK:= qrFreq > 0, Q=> );
rtrig_ixEmergencyStop(CLK:= ixEmergencyStop, Q=> );
rtrig_ixReset(CLK:= ixReset, Q=> );
rtrig_ixStarted(CLK:= ixStarted, Q=> );
rtrig_ixStopped(CLK:= ixStopped, Q=> );

ProcessErrorHandling();
ProcessFrequencyControl();
ProcessSignal();
ProcessTimers();
                  

METHOD cmdReset : BOOL
VAR_INPUT
END_VAR
                          qxEmergencyStopStatus := FALSE;
qxErrorInvalidInaccuracy := FALSE;
qxErrorDevice := FALSE;
qxDelayError := FALSE;
xErrorFixation := FALSE;

                        
END_METHOD

METHOD cmdStart : BOOL
VAR_INPUT
	xStart : BOOL;
END_VAR
                          IF xStart THEN
	qxStart := TRUE;
END_IF;

IF NOT xStart THEN
	qxStart := FALSE;
END_IF;
                        
END_METHOD

METHOD cmdFastStart : BOOL
VAR_INPUT
	xStart : BOOL;
END_VAR
                          IF xStart THEN
	cmdStart(TRUE);
	qrFreq := iqrSetFreq;
END_IF;
                        
END_METHOD

METHOD cmdStop : BOOL
VAR_INPUT
	xStop : BOOL;
END_VAR
                          IF xStop THEN
	qxStop := TRUE;
END_IF;

IF NOT xStop THEN
	qxStop := FALSE;
END_IF;
                        
END_METHOD

METHOD cmdEmergencyStop : BOOL
VAR_INPUT
	xStop : BOOL;
END_VAR
                          IF xStop THEN
	cmdStop(TRUE);
	qxEmergencyStopStatus := TRUE;
END_IF;
                        
END_METHOD

METHOD GetErrorInvalidInaccuracy : BOOL
VAR_INPUT
END_VAR
                          GetErrorInvalidInaccuracy := NOT CheckFrequencyInaccuracy();
                        
END_METHOD

METHOD GetErrorDevice : BOOL
VAR_INPUT
END_VAR
                          GetErrorDevice := ixDeviceError;
                        
END_METHOD

METHOD GetDelayError : BOOL
VAR_INPUT
END_VAR
                          GetDelayError := (ton_StopDisable.Q AND NOT qxEmergencyStopStatus) OR ton_StartDisable.Q;
                        
END_METHOD

METHOD UpdateStatus : BOOL
VAR_INPUT
END_VAR
                          qxStartStatus := qxStart;
qxStopStatus := qxStop;

// Обновление статуса аварийной остановки по сигналу кнопки
IF rtrig_ixEmergencyStop.Q THEN qxEmergencyStopStatus := TRUE; END_IF;

// Остановка рабочего процесса по сигналу заднего фронта qrFreq > 0
IF ftrig_StopWorkProcess.Q THEN xWorkProcess := FALSE; END_IF;

// Остановка рабочего процесса xWorkProcess AND qrFreq = 0 по таймеру
IF ton_stopWorkProcess.Q THEN xWorkProcess := FALSE; END_IF;
                        
END_METHOD

METHOD CalculateNewFrequency  : REAL
VAR_INPUT
END_VAR
                          IF iqrSetFreq + irUpdateCycleStep < qrFreq THEN
	CalculateNewFrequency := qrFreq - irUpdateCycleStep;
ELSIF iqrSetFreq - irUpdateCycleStep > qrFreq THEN
	CalculateNewFrequency := qrFreq + irUpdateCycleStep;
ELSE
	CalculateNewFrequency := iqrSetFreq;
END_IF;
                        
END_METHOD

METHOD CheckFrequencyInaccuracy : BOOL
VAR_INPUT
END_VAR
                          IF irActualFreq < qrFreq THEN
	CheckFrequencyInaccuracy := qrFreq - irActualFreq <= irActualFreqInaccuracy;
ELSIF irActualFreq > qrFreq THEN
	CheckFrequencyInaccuracy :=irActualFreq - qrFreq <= irActualFreqInaccuracy;
ELSIF irActualFreq = qrFreq THEN
	CheckFrequencyInaccuracy := TRUE;
ELSE
	CheckFrequencyInaccuracy := FALSE;
END_IF;


                        
END_METHOD

METHOD ShouldUpdateFrequency  : BOOL
VAR_INPUT
END_VAR
                          ShouldUpdateFrequency := iqrSetFreq <> qrFreq 
	AND CheckFrequencyInaccuracy()
	AND rtrig_updateCycle.Q
	AND NOT xErrorFixation
	AND ixDeviceReady
	AND NOT qxEmergencyStopStatus
	AND (iqrSetFreq <= irMaxFreq) 
	AND (iqrSetFreq >= 0);
                        
END_METHOD

METHOD ProcessTimers : BOOL
VAR_INPUT
END_VAR
                          // Таймер для цикла обновления
blink_updateCycle(
    ENABLE:= xWorkProcess, 
    TIMELOW:= itUpdateCycle, 
    TIMEHIGH:= T#100MS
);
rtrig_updateCycle(CLK:= blink_updateCycle.OUT, Q=> );

// Таймер остановки рабочего процесса
ton_stopWorkProcess(
    IN:= xWorkProcess AND qrFreq = 0, 
    PT:= T#5S
);

ton_StopDisable(
	IN:= qxStop, 
	PT:= itStartStopDelay, 
	Q=> , 
	ET=> );

ton_StartDisable(
	IN:= qxStart, 
	PT:= itStartStopDelay,
	Q=> , 
	ET=> );
                        
END_METHOD

METHOD ProcessErrorHandling : BOOL
VAR_INPUT
END_VAR
                          // Обобщённая фиксация всех ошибок в одну переменную
IF GetErrorDevice() OR GetErrorInvalidInaccuracy() OR rtrig_ixEmergencyStop.Q THEN
	xErrorFixation := TRUE;
END_IF;

IF GetErrorDevice() THEN qxErrorDevice := TRUE; END_IF;
IF GetErrorInvalidInaccuracy() THEN qxErrorInvalidInaccuracy := TRUE; END_IF;
IF GetDelayError() THEN qxDelayError := TRUE; END_IF;
                        
END_METHOD

METHOD ProcessFrequencyControl : BOOL
VAR_INPUT
END_VAR
                          // Плавное изменение частоты
IF ShouldUpdateFrequency() THEN
    qrFreq := CalculateNewFrequency();
END_IF;

// Защита от задания частоты вне диапазона
IF iqrSetFreq > irMaxFreq THEN iqrSetFreq := irMaxFreq; END_IF;
IF iqrSetFreq < 0 THEN iqrSetFreq := 0; END_IF;

// Задание частоты на 0 при получении сигнала остановки
IF rtrig_ixStop.Q AND NOT ixSmoothStop THEN qrFreq := 0; END_IF;
                        
END_METHOD

METHOD ProcessSignal : BOOL
VAR_INPUT
END_VAR
                          UpdateStatus();

// Обработка сигнала старт
IF rtrig_ixStart.Q OR rtrig_ixFastStart.Q THEN 
	cmdStart(TRUE); 
	cmdStop(FALSE); 
	xWorkProcess := TRUE;
END_IF;
// Завершение сигнала старт
IF rtrig_ixStarted.Q OR ton_StartDisable.Q THEN 
	cmdStart(FALSE);
END_IF;

// Отработка сигнала стоп
IF rtrig_ixStop.Q THEN 
	cmdStop(TRUE); 
	cmdStart(FALSE); 
	xWorkProcess := TRUE;
END_IF;
// Завершение сигнала стоп
IF rtrig_ixStopped.Q OR ton_StopDisable.Q THEN 
	cmdStop(FALSE); 
END_IF;

// Обработка сигнала аварийной остановки
IF rtrig_ixEmergencyStop.Q THEN
	cmdStop(TRUE);
END_IF;

// Обработка сигнала сброса ошибок
IF rtrig_ixReset.Q THEN
	cmdReset();
END_IF;

// Обработка сигнала быстрого старта
IF rtrig_ixFastStart.Q THEN
	cmdFastStart(TRUE);
END_IF;
                        
END_METHOD
END_FUNCTION_BLOCK

PROGRAM MAIN
VAR
	// 	== ДЛЯ ТЕСТА, ПОТОМ УДАЛИТЬ ==

	PLC_Mode : INT := 0; // 0 – «Авто», 1 – «Обрыв связи», 2 – «Местный-Сервис»
	
	// LeftSide Маска входов ПЛК
	_0303_05_PU01_ixKM_StatusOn : BOOL;				// Контактор ПРЯМ. ПУСК Насос 0303.05-PU-01
	_0303_05_PU01_ixKM_VFD_StatusOn : BOOL;			// Контактор ПРЯМ. ЧРП Насос 0303.05-PU-01
	_0303_05_PU02_ixKM_StatusOn : BOOL;				// Контактор ПРЯМ. ПУСК Насос 0303.05-PU-02
	_0303_05_PU02_ixKM_VFD_StatusOn : BOOL;			// Контактор ПРЯМ. ЧРП Насос 0303.05-PU-02
	_0303_05_PU03_ixKM_StatusOn : BOOL;				// Контактор ПРЯМ. ПУСК Насос 0303.05-PU-03
	_0303_05_PU03_ixKM_VFD_StatusOn : BOOL;			// Контактор ПРЯМ. ЧРП Насос 0303.05-PU-03
	_0303_05_PU04_ixKM_StatusOn : BOOL;				// Контактор ПРЯМ. ПУСК Насос 0303.05-PU-04
	_0303_05_PU04_ixKM_VFD_StatusOn : BOOL;			// Контактор ПРЯМ. ЧРП Насос 0303.05-PU-04
	_0303_05_PU05_ixKM_StatusOn : BOOL;				// Контактор ПРЯМ. ПУСК Насос 0303.05-PU-05
	_0303_05_PU05_ixKM_VFD_StatusOn : BOOL;			// Контактор ПРЯМ. ЧРП Насос 0303.05-PU-05
	_0303_05_BY08_ixShutter_PosOpen : BOOL;			// Положение ОТКР. Затвор 0303.05-BY-08
	_0303_05_BY08_ixShutter_PosClosed : BOOL;		// Положение ЗАКР. Затвор 0303.05-BY-08
	
	// RightSide Маска выходов ПЛК
	_0303_05_qxEmergencyStop : BOOL;			// Реле аварийного останова
	_0303_05_PU01_qxDryRun : BOOL;				// Насос 0303.05-PU-01 Сухой ход
	_0303_05_PU02_qxDryRun : BOOL;				// Насос 0303.05-PU-02 Сухой ход
	_0303_05_PU03_qxDryRun : BOOL;				// Насос 0303.05-PU-03 Сухой ход
	_0303_05_PU04_qxDryRun : BOOL;				// Насос 0303.05-PU-04 Сухой ход
	_0303_05_PU05_qxDryRun : BOOL;				// Насос 0303.05-PU-05 Сухой ход
	_0303_05_1KM8_qxOn : BOOL;					// Включить 1KM8
	_0303_05_2KM8_qxOn : BOOL;					// Включить 2KM8
	
	// 	==============================================
	
	// Общие глобальные переменные
	tRattlingDelay : TIME := T#100MS;			// Задержка получения сигнала входов (защита от дребезга)
	vfd_iChange : INT;							// Выбор работающего ЧРП
	pu_iChange : INT;							// Выбор насоса для исполнения команд
	by_iChange : INT;							// Выбор затвора для исполнения команд
	// VFD
	// Конфигурация
	vfd_rMaxFreq : REAL := 50;					// Максимальное задание частоты
	vfd_tUpdateCycle : TIME := T#2S;			// Время обновления цикла плавного пуска/остановки в TIME
	vfd_rUpdateCycleStep : REAL := 1.5;			// Шаг обновления частоты за 1 цикл
	vfd_rActualFreqInaccuracy : REAL := 0.2;	// Максимальная допустимая погрешность для ЧРП
	vfd_tStartStopDelay : TIME := T#10S;		// Время задержки сигнала старт и стоп до его отключения и выхода ошибки долгого ожидания отклика механизма
	vfd_xReserveStatus : BOOL;					// true - замена основного ЧРП на резерв
	// Общие переменные
	vfd_rSetFreq : REAL;						// Задание частоты
	// ЧРП Основной
	VFD_MAIN : FB_VFD_CTRL;
	 // ЧРП Резерв
	VFD_RESERVE : FB_VFD_CTRL;
	
	// init_ServiceAutoSignals (команды режима сервис и авто)
	xPU_Start 			: FB_SignalSplit;
	xPU_Stop 			: FB_SignalSplit;
	xPU_Reset 			: FB_SignalSplit;
	xPU_Change_VFDtoBP	: FB_SignalSplit;
	xPU_Change_BPtoVFD	: FB_SignalSplit;

	xVFD_Start          : FB_SignalSplit;
	xVFD_Stop           : FB_SignalSplit;
	xVFD_EmergencyStop	: FB_SignalSplit;
	xVFD_Reset			: FB_SignalSplit;
	
	xBY_Open			: FB_SignalSplit;
	xBY_Close           : FB_SignalSplit;
	xBY_Stop            : FB_SignalSplit;
	xBY_Reset           : FB_SignalSplit;
	
	
	// **Process_BY_Commands**
	rtrig_byCmd_xOpen 				: R_TRIG;
	rtrig_byCmd_xClose             	: R_TRIG;
	rtrig_byCmd_xStop     			: R_TRIG;
	rtrig_byCmd_xReset              : R_TRIG;
	
	// **Process_PU_Commands**
	rtrig_puCmd_xStart 				: R_TRIG;
	rtrig_puCmd_xStop               : R_TRIG;
	rtrig_puCmd_xReset              : R_TRIG;
	rtrig_puCmd_xChange_VFDtoBP     : R_TRIG;
	rtrig_puCmd_xChange_BPtoVFD     : R_TRIG;
	
	// **Process_VFD_Commands**
	rtrig_vfdCmd_xStart				: R_TRIG;
	rtrig_vfdCmd_xStop              : R_TRIG;
	rtrig_vfdCmd_xEmergencyStop		: R_TRIG;
	rtrig_vfdCmd_xReset             : R_TRIG;
	
	// ЗРА
	
	BY1		: FB_Shutter;
	BY2     : FB_Shutter;
	BY3     : FB_Shutter;
	BY4     : FB_Shutter;
	BY5     : FB_Shutter;
	BY7     : FB_Shutter;
	BY8     : FB_Shutter;
	
	
	// Дребезг сигналов
	in_0303_05_1_ixSection1_OverheatAlarm          : INPUT_OUTPUT;
	in_0303_05_1_ixSection1_OverheatWarning        : INPUT_OUTPUT;
	in_0303_05_1_ixVFD_Failure                     : INPUT_OUTPUT;
	in_0303_05_1_ixVFD_InWork                      : INPUT_OUTPUT;
	in_0303_05_1_ixVFD_Manual                      : INPUT_OUTPUT;
	in_0303_05_1_ixVFD_Ready                       : INPUT_OUTPUT;
	in_0303_05_2_ixSection1_OverheatAlarm          : INPUT_OUTPUT;
	in_0303_05_2_ixSection1_OverheatWarning        : INPUT_OUTPUT;
	in_0303_05_2_ixVFD_Failure                     : INPUT_OUTPUT;
	in_0303_05_2_ixVFD_InWork                      : INPUT_OUTPUT;
	in_0303_05_2_ixVFD_Manual                      : INPUT_OUTPUT;
	in_0303_05_2_ixVFD_Ready                       : INPUT_OUTPUT;
	in_0303_05_1KM8_ixStatusOn                     : INPUT_OUTPUT;
	in_0303_05_2KM8_ixStatusOn                     : INPUT_OUTPUT;
	in_0303_05_BY01_ixKM_PosClosed                 : INPUT_OUTPUT;
	in_0303_05_BY01_ixKM_PosOpen                   : INPUT_OUTPUT;
	in_0303_05_BY01_ixShutter_PosClosed            : INPUT_OUTPUT;
	in_0303_05_BY01_ixShutter_PosOpen              : INPUT_OUTPUT;
	in_0303_05_BY01_ixShutter_StatusError          : INPUT_OUTPUT;
	in_0303_05_BY01_ixShutter_StatusReady          : INPUT_OUTPUT;
	in_0303_05_BY02_ixKM_PosClosed                 : INPUT_OUTPUT;
	in_0303_05_BY02_ixKM_PosOpen                   : INPUT_OUTPUT;
	in_0303_05_BY02_ixShutter_PosClosed            : INPUT_OUTPUT;
	in_0303_05_BY02_ixShutter_PosOpen              : INPUT_OUTPUT;
	in_0303_05_BY02_ixShutter_StatusError          : INPUT_OUTPUT;
	in_0303_05_BY02_ixShutter_StatusReady          : INPUT_OUTPUT;
	in_0303_05_BY03_ixKM_PosClosed                 : INPUT_OUTPUT;
	in_0303_05_BY03_ixKM_PosOpen                   : INPUT_OUTPUT;
	in_0303_05_BY03_ixShutter_PosClosed            : INPUT_OUTPUT;
	in_0303_05_BY03_ixShutter_PosOpen              : INPUT_OUTPUT;
	in_0303_05_BY03_ixShutter_StatusError          : INPUT_OUTPUT;
	in_0303_05_BY03_ixShutter_StatusReady          : INPUT_OUTPUT;
	in_0303_05_BY04_ixKM_PosClosed                 : INPUT_OUTPUT;
	in_0303_05_BY04_ixKM_PosOpen                   : INPUT_OUTPUT;
	in_0303_05_BY04_ixShutter_PosClosed            : INPUT_OUTPUT;
	in_0303_05_BY04_ixShutter_PosOpen              : INPUT_OUTPUT;
	in_0303_05_BY04_ixShutter_StatusError          : INPUT_OUTPUT;
	in_0303_05_BY04_ixShutter_StatusReady          : INPUT_OUTPUT;
	in_0303_05_BY05_ixKM_PosClosed                 : INPUT_OUTPUT;
	in_0303_05_BY05_ixKM_PosOpen                   : INPUT_OUTPUT;
	in_0303_05_BY05_ixShutter_PosClosed            : INPUT_OUTPUT;
	in_0303_05_BY05_ixShutter_PosOpen              : INPUT_OUTPUT;
	in_0303_05_BY05_ixShutter_StatusError          : INPUT_OUTPUT;
	in_0303_05_BY05_ixShutter_StatusReady          : INPUT_OUTPUT;
	in_0303_05_BY07_ixKM_PosClosed                 : INPUT_OUTPUT;
	in_0303_05_BY07_ixKM_PosOpen                   : INPUT_OUTPUT;
	in_0303_05_BY07_ixShutter_PosClosed            : INPUT_OUTPUT;
	in_0303_05_BY07_ixShutter_PosOpen              : INPUT_OUTPUT;
	in_0303_05_BY07_ixShutter_StatusError          : INPUT_OUTPUT;
	in_0303_05_BY07_ixShutter_StatusReady          : INPUT_OUTPUT;
	in_0303_05_BY08_ixKM_PosClosed                 : INPUT_OUTPUT;
	in_0303_05_BY08_ixKM_PosOpen                   : INPUT_OUTPUT;
	in_0303_05_BY08_ixShutter_PosClosed            : INPUT_OUTPUT;
	in_0303_05_BY08_ixShutter_PosOpen              : INPUT_OUTPUT;
	in_0303_05_BY08_ixShutter_StatusError          : INPUT_OUTPUT;
	in_0303_05_BY08_ixShutter_StatusReady          : INPUT_OUTPUT;
	in_0303_05_PU01_ixKM_StatusManualStart         : INPUT_OUTPUT;
	in_0303_05_PU01_ixKM_StatusManualStop          : INPUT_OUTPUT;
	in_0303_05_PU01_ixKM_StatusOn                  : INPUT_OUTPUT;
	in_0303_05_PU01_ixKM_VFD_StatusOn              : INPUT_OUTPUT;
	in_0303_05_PU01_ixStatusManual                 : INPUT_OUTPUT;
	in_0303_05_PU02_ixKM_StatusManualStart         : INPUT_OUTPUT;
	in_0303_05_PU02_ixKM_StatusManualStop          : INPUT_OUTPUT;
	in_0303_05_PU02_ixKM_StatusOn                  : INPUT_OUTPUT;
	in_0303_05_PU02_ixKM_VFD_StatusOn              : INPUT_OUTPUT;
	in_0303_05_PU02_ixStatusManual                 : INPUT_OUTPUT;
	in_0303_05_PU03_ixKM_StatusManualStart         : INPUT_OUTPUT;
	in_0303_05_PU03_ixKM_StatusManualStop          : INPUT_OUTPUT;
	in_0303_05_PU03_ixKM_StatusOn                  : INPUT_OUTPUT;
	in_0303_05_PU03_ixKM_VFD_StatusOn              : INPUT_OUTPUT;
	in_0303_05_PU03_ixStatusManual                 : INPUT_OUTPUT;
	in_0303_05_PU04_ixKM_StatusManualStart         : INPUT_OUTPUT;
	in_0303_05_PU04_ixKM_StatusManualStop          : INPUT_OUTPUT;
	in_0303_05_PU04_ixKM_StatusOn                  : INPUT_OUTPUT;
	in_0303_05_PU04_ixKM_VFD_StatusOn              : INPUT_OUTPUT;
	in_0303_05_PU04_ixStatusManual                 : INPUT_OUTPUT;
	in_0303_05_PU05_ixKM_StatusManualStart         : INPUT_OUTPUT;
	in_0303_05_PU05_ixKM_StatusManualStop          : INPUT_OUTPUT;
	in_0303_05_PU05_ixKM_StatusOn                  : INPUT_OUTPUT;
	in_0303_05_PU05_ixKM_VFD_StatusOn              : INPUT_OUTPUT;
	in_0303_05_PU05_ixStatusManual                 : INPUT_OUTPUT;
END_VAR

                    Initialization();

Process_VFD();

Process_PU();
                  

METHOD Init_VFD_Main
VAR_INPUT
END_VAR
                          VFD_MAIN(
	irMaxFreq:= vfd_rMaxFreq, 
	itUpdateCycle:= vfd_tUpdateCycle, 
	irUpdateCycleStep:= vfd_rUpdateCycleStep, 
	irActualFreqInaccuracy:= vfd_rActualFreqInaccuracy, 
	ixSmoothStop:= , 
	itStartStopDelay:= vfd_tStartStopDelay, 
	ixStart:= , 
	ixFastStart:= , 
	ixStop:= , 
	ixEmergencyStop:= , 
	ixReset:= , 
	ixStarted:= GetStatus_PU_VFD(pu_iChange), 
	ixStopped:= NOT GetStatus_PU_VFD(pu_iChange), 
	ixDeviceError:= GetStatus_VFD_Error(1), 
	ixDeviceReady:= GetStatus_VFD_Ready(1), 
	irActualFreq:= GetStatus_VFD_ActualFreq(1), 
	qrFreq=> , 
	qxStart=> , 
	qxStop=> , 
	qxStartStatus=> , 
	qxStopStatus=> , 
	qxEmergencyStopStatus=> , 
	qxErrorInvalidInaccuracy=> , 
	qxErrorDevice=> , 
	qxDelayError=> , 
	iqrSetFreq:= vfd_rSetFreq);
                        
END_METHOD

METHOD Init_VFD_Reserve
VAR_INPUT
END_VAR
                          VFD_RESERVE(
	irMaxFreq:= vfd_rMaxFreq, 
	itUpdateCycle:= vfd_tUpdateCycle, 
	irUpdateCycleStep:= vfd_rUpdateCycleStep, 
	irActualFreqInaccuracy:= vfd_rActualFreqInaccuracy, 
	ixSmoothStop:= , 
	itStartStopDelay:= vfd_tStartStopDelay, 
	ixStart:= , 
	ixFastStart:= , 
	ixStop:= , 
	ixEmergencyStop:= , 
	ixReset:= , 
	ixStarted:= GetStatus_PU_VFD(pu_iChange), 
	ixStopped:= NOT GetStatus_PU_VFD(pu_iChange), 
	ixDeviceError:= GetStatus_VFD_Error(2), 
	ixDeviceReady:= GetStatus_VFD_Ready(2), 
	irActualFreq:= GetStatus_VFD_ActualFreq(2), 
	qrFreq=> , 
	qxStart=> , 
	qxStop=> , 
	qxStartStatus=> , 
	qxStopStatus=> , 
	qxEmergencyStopStatus=> , 
	qxErrorInvalidInaccuracy=> , 
	qxErrorDevice=> , 
	qxDelayError=> , 
	iqrSetFreq:= vfd_rSetFreq);
                        
END_METHOD

